	{attribute 'TcIecLibraryType'}
	{attribute 'external_name' := 'F_VN_StartAbsWatchdog_GUID_CDB36576_3437_07D6_675F_669467F27649'}
	(* Starts a cooperative watchdog given an absolute stop time. *)
	FUNCTION F_VN_StartAbsWatchdog : HRESULT
	VAR_INPUT
		tStop	:	DINT;	(* Stop time in us *)
		hrPrev	:	HRESULT;	(* HRESULT indicating the result of previous operations (If SUCCEEDED(hrPrev) equals false, no operation is executed.) *)
	END_VAR

END_FUNCTION

// Functions/Control Functions/F_VN_StartAbsWatchdogExp

	{attribute 'TcIecLibraryType'}
	{attribute 'external_name' := 'F_VN_StartAbsWatchdogExp_GUID_5DF99523_737E_0B42_4AEA_F8C27544139F'}
	(* Start a cooperative watchdog given an absolute stop time. (expert function) *)
	FUNCTION F_VN_StartAbsWatchdogExp : HRESULT
	VAR_INPUT
		tStop	:	DINT;	(* Stop time in us *)
		eWatchdogAccType	:	ETcWatchdogAccumulationType;	(* Accumalation method used for combining the results of multiple functions enclosed by this watchdog *)
		hrPrev	:	HRESULT;	(* HRESULT indicating the result of previous operations (If SUCCEEDED(hrPrev) equals false, no operation is executed.) *)
	END_VAR

END_FUNCTION

// Functions/Control Functions/F_VN_StartRelWatchdog

	{attribute 'TcIecLibraryType'}
	{attribute 'external_name' := 'F_VN_StartRelWatchdog_GUID_36307EEF_0607_0986_40C6_26A6AD435D06'}
	(* Starts a cooperative watchdog given a stop time relative to the current time. *)
	FUNCTION F_VN_StartRelWatchdog : HRESULT
	VAR_INPUT
		tStop	:	DINT;	(* Stop time in us *)
		hrPrev	:	HRESULT;	(* HRESULT indicating the result of previous operations (If SUCCEEDED(hrPrev) equals false, no operation is executed.) *)
	END_VAR

END_FUNCTION

// Functions/Control Functions/F_VN_StartRelWatchdogExp

	{attribute 'TcIecLibraryType'}
	{attribute 'external_name' := 'F_VN_StartRelWatchdogExp_GUID_3570B399_84A1_03B6_6569_A22DA832851F'}
	(* Start a cooperative watchdog given a stop time relative to the current time. (expert function) *)
	FUNCTION F_VN_StartRelWatchdogExp : HRESULT
	VAR_INPUT
		tStop	:	DINT;	(* Stop time in us *)
		eWatchdogAccType	:	ETcWatchdogAccumulationType;	(* Accumalation method used for combining the results of multiple functions enclosed by this watchdog *)
		hrPrev	:	HRESULT;	(* HRESULT indicating the result of previous operations (If SUCCEEDED(hrPrev) equals false, no operation is executed.) *)
	END_VAR

END_FUNCTION

// Functions/Control Functions/F_VN_StopWatchdog

	{attribute 'TcIecLibraryType'}
	{attribute 'external_name' := 'F_VN_StopWatchdog_GUID_5FE8103F_689C_0837_5C85_B4C88911468C'}
	(* Stops a watchdog and provide runtime information. *)
	FUNCTION F_VN_StopWatchdog : HRESULT
	VAR_INPUT
		hrStartWatchdog	:	HRESULT;	(* HRESULT indicating the result of the function used to start the watchdog (If SUCCEEDED(hrStartWatchdog) equals false, no operation is executed.) *)
	END_VAR
	VAR_OUTPUT
		nFunctionsMonitored	:	ULINT;	(* Returns the number of functions monitored *)
		nFractionProcessed	:	UDINT;	(* Returns the fraction processed accumulated over the monitored functions in percent *)
		tRest	:	DINT;	(* Returns the remaining computation time in us (may be negative) *)
	END_VAR

END_FUNCTION

// Functions/Image Segmentation/F_VN_AdaptiveThreshold

	{attribute 'TcIecLibraryType'}
	{attribute 'external_name' := 'F_VN_AdaptiveThreshold_GUID_B1BC4894_E3E4_011A_5395_9D7E3F472C15'}
	(* Apply an adaptive threshold to a gray level image. *)
	FUNCTION F_VN_AdaptiveThreshold : HRESULT
	VAR_INPUT
		ipSrcImage	:	ITcVnImage;	(* Source image (1 channel, elements of type USINT) *)
		ipDestImage	:	REFERENCE TO ITcVnImage;	(* Destination image (An appropriate destination image will be created if required.) *)
		fMaxValue	:	LREAL;	(* Value assigned to pixels for which the threshold condition is true *)
		hrPrev	:	HRESULT;	(* HRESULT indicating the result of previous operations (If SUCCEEDED(hrPrev) equals false, no operation is executed.) *)
	END_VAR

END_FUNCTION

// Functions/Image Segmentation/F_VN_AdaptiveThresholdExp

	{attribute 'TcIecLibraryType'}
	{attribute 'external_name' := 'F_VN_AdaptiveThresholdExp_GUID_E41ECDB8_1C09_051C_54A7_3EA4088C1F31'}
	(* Apply an adaptive threshold to a gray level image. (expert function) *)
	FUNCTION F_VN_AdaptiveThresholdExp : HRESULT
	VAR_INPUT
		ipSrcImage	:	ITcVnImage;	(* Source image (1 channel, elements of type USINT) *)
		ipDestImage	:	REFERENCE TO ITcVnImage;	(* Destination image (An appropriate destination image will be created if required.) *)
		fMaxValue	:	LREAL;	(* Value assigned to pixels for which the threshold condition is true *)
		eAdaptiveMethod	:	ETcVnAdaptiveThresholdMethod;	(* Adaptive threshold method to be applied (MEAN: threshold value will be calculated as a mean of the nBlockSize x nBlockSize neighborhood of (x,y) minus fConstant. GAUSSIAN: threshold value is a weighted sum (cross-correlation with a Gaussian window) of the nBlockSize x nBlockSize neighborhood of (x,y) minus fConstant. *)
		eThresholdType	:	ETcVnThresholdType;	(* Threshold type to be applied (only BINARY and BINARY_INV are supported) *)
		nBlockSize	:	UDINT;	(* Size of the pixel neighborhood to calculate the local threshold (3, 5, 7, ...) *)
		fConstant	:	LREAL;	(* Constant that is subtracted from the weighted mean of the pixel neighborhood, which leads to the local threshold *)
		hrPrev	:	HRESULT;	(* HRESULT indicating the result of previous operations (If SUCCEEDED(hrPrev) equals false, no operation is executed.) *)
	END_VAR

END_FUNCTION

// Functions/Image Segmentation/F_VN_CheckColorRange

	{attribute 'TcIecLibraryType'}
	{attribute 'external_name' := 'F_VN_CheckColorRange_GUID_5F05A5F1_5853_0BB7_40B0_9B84FD8E7D5D'}
	(* Check if the pixel values of an image lie in a given range. The destination image has the same size as the source image but only one channel with
          a pixel element size of 8 bit. Its elements are set to 255 if the corresponding pixels of the source image are in the checked range and set to 0 otherwise. *)
	FUNCTION F_VN_CheckColorRange : HRESULT
	VAR_INPUT
		ipSrcImage	:	ITcVnImage;	(* Source image *)
		ipDestImage	:	REFERENCE TO ITcVnImage;	(* Destination image (An appropriate destination image will be created if required.) *)
		aLowerBounds	:	REFERENCE TO TcVnVector4_LREAL;	(* Channel-wise lower bounds (Unused channels are ignored.) *)
		aUpperBounds	:	REFERENCE TO TcVnVector4_LREAL;	(* Channel-wise upper bounds (Unused channels are ignored.) *)
		hrPrev	:	HRESULT;	(* HRESULT indicating the result of previous operations (If SUCCEEDED(hrPrev) equals false, no operation is executed.) *)
	END_VAR

END_FUNCTION

// Functions/Image Segmentation/F_VN_Threshold

	{attribute 'TcIecLibraryType'}
	{attribute 'external_name' := 'F_VN_Threshold_GUID_F4BFB9FB_0241_0ABA_6497_302E4CB6A3F0'}
	(* Apply a fixed threshold or a dynamic threshold according to Otsu. *)
	FUNCTION F_VN_Threshold : HRESULT
	VAR_INPUT
		ipSrcImage	:	ITcVnImage;	(* Source image (For Otsu and Triangle threshold types, only 1 channel of TCVN_ET_USINT is supported) *)
		ipDestImage	:	REFERENCE TO ITcVnImage;	(* Destination image (An appropriate destination image will be created if required.) *)
		fThreshold	:	LREAL;	(* Fixed threshold (unused if dynamic thresholding is selected) *)
		fMaxValue	:	LREAL;	(* Maximum pixel value *)
		eThresholdType	:	ETcVnThresholdType;	(* Threshold type to be applied *)
		hrPrev	:	HRESULT;	(* HRESULT indicating the result of previous operations (If SUCCEEDED(hrPrev) equals false, no operation is executed.) *)
	END_VAR

END_FUNCTION

// Functions/Image Segmentation/F_VN_WatershedSegmentationExp

	{attribute 'TcIecLibraryType'}
	{attribute 'external_name' := 'F_VN_WatershedSegmentationExp_GUID_05447CF8_8CF8_0191_6A21_DD063D69ABC3'}
	(* Apply a marker-based watershed segmentation. (expert function) *)
	FUNCTION F_VN_WatershedSegmentationExp : HRESULT
	VAR_INPUT
		ipSrcImage	:	ITcVnImage;	(* Source image (USINT, 3 channels) *)
		ipDestImage	:	REFERENCE TO ITcVnImage;	(* Destination image (DINT, 1 channel. An appropriate image will be created if required.) *)
		ipMarkers	:	ITcVnImage;	(* Marker image (DINT, 1 channel) *)
		hrPrev	:	HRESULT;	(* HRESULT indicating the result of previous operations (If SUCCEEDED(hrPrev) equals false, no operation is executed.) *)
	END_VAR

END_FUNCTION

// Functions/Algebraic Container Operations/F_VN_AddContainers

	{attribute 'TcIecLibraryType'}
	{attribute 'external_name' := 'F_VN_AddContainers_GUID_34C85C3E_C161_0A16_51C0_0BD519308179'}
	(* Element-wise addition of two containers (same length and type). *)
	FUNCTION F_VN_AddContainers : HRESULT
	VAR_INPUT
		ipSrcContainer1	:	ITcVnContainer;	(* Source container 1 *)
		ipSrcContainer2	:	ITcVnContainer;	(* Source container 2 *)
		ipDestContainer	:	REFERENCE TO ITcVnContainer;	(* Returns the resulting container *)
		hrPrev	:	HRESULT;	(* HRESULT indicating the result of previous operations (If SUCCEEDED(hrPrev) equals false, no operation is executed.) *)
	END_VAR

END_FUNCTION

// Functions/Algebraic Container Operations/F_VN_BitwiseAndContainers

	{attribute 'TcIecLibraryType'}
	{attribute 'external_name' := 'F_VN_BitwiseAndContainers_GUID_EB7545F4_E7C1_0AC8_4065_DD74452EA045'}
	(* Element-wise application of a bit-wise AND operator to two containers (same length and type, integer only). *)
	FUNCTION F_VN_BitwiseAndContainers : HRESULT
	VAR_INPUT
		ipSrcContainer1	:	ITcVnContainer;	(* Source container 1 *)
		ipSrcContainer2	:	ITcVnContainer;	(* Source container 2 *)
		ipDestContainer	:	REFERENCE TO ITcVnContainer;	(* Returns the resulting container *)
		hrPrev	:	HRESULT;	(* HRESULT indicating the result of previous operations (If SUCCEEDED(hrPrev) equals false, no operation is executed.) *)
	END_VAR

END_FUNCTION

// Functions/Algebraic Container Operations/F_VN_BitwiseNotContainer

	{attribute 'TcIecLibraryType'}
	{attribute 'external_name' := 'F_VN_BitwiseNotContainer_GUID_F7145E10_2EC4_02FB_47B2_0962C0E72D64'}
	(* Element-wise application of a bit-wise NOT operator to a container (integer only). *)
	FUNCTION F_VN_BitwiseNotContainer : HRESULT
	VAR_INPUT
		ipSrcContainer	:	ITcVnContainer;	(* Source container *)
		ipDestContainer	:	REFERENCE TO ITcVnContainer;	(* Returns the resulting container *)
		hrPrev	:	HRESULT;	(* HRESULT indicating the result of previous operations (If SUCCEEDED(hrPrev) equals false, no operation is executed.) *)
	END_VAR

END_FUNCTION

// Functions/Algebraic Container Operations/F_VN_BitwiseOrContainers

	{attribute 'TcIecLibraryType'}
	{attribute 'external_name' := 'F_VN_BitwiseOrContainers_GUID_F073C4C8_8568_027C_57D8_3DAA401B2897'}
	(* Element-wise application of a bit-wise OR operator to two containers (same length and type, integer only). *)
	FUNCTION F_VN_BitwiseOrContainers : HRESULT
	VAR_INPUT
		ipSrcContainer1	:	ITcVnContainer;	(* Source container 1 *)
		ipSrcContainer2	:	ITcVnContainer;	(* Source container 2 *)
		ipDestContainer	:	REFERENCE TO ITcVnContainer;	(* Returns the resulting container *)
		hrPrev	:	HRESULT;	(* HRESULT indicating the result of previous operations (If SUCCEEDED(hrPrev) equals false, no operation is executed.) *)
	END_VAR

END_FUNCTION

// Functions/Algebraic Container Operations/F_VN_BitwiseXorContainers

	{attribute 'TcIecLibraryType'}
	{attribute 'external_name' := 'F_VN_BitwiseXorContainers_GUID_B00A3AA9_EBBD_07B2_4D65_1CE7DD68EA4F'}
	(* Element-wise application of a bit-wise XOR operator to two containers (same length and type, integer only). *)
	FUNCTION F_VN_BitwiseXorContainers : HRESULT
	VAR_INPUT
		ipSrcContainer1	:	ITcVnContainer;	(* Source container 1 *)
		ipSrcContainer2	:	ITcVnContainer;	(* Source container 2 *)
		ipDestContainer	:	REFERENCE TO ITcVnContainer;	(* Returns the resulting container *)
		hrPrev	:	HRESULT;	(* HRESULT indicating the result of previous operations (If SUCCEEDED(hrPrev) equals false, no operation is executed.) *)
	END_VAR

END_FUNCTION

// Functions/Algebraic Container Operations/F_VN_DivideContainers

	{attribute 'TcIecLibraryType'}
	{attribute 'external_name' := 'F_VN_DivideContainers_GUID_4F7AC07C_47AD_08DA_5AD8_2625E1B3B314'}
	(* Element-wise division of two containers (same length and type). In case of integer division by zero, the resulting element is set to 0 and S_DIVISION_BY_ZERO is returned instead of S_OK (value can be changed in F_VN_DivideContainersExp). *)
	FUNCTION F_VN_DivideContainers : HRESULT
	VAR_INPUT
		ipSrcContainer1	:	ITcVnContainer;	(* Source container 1 *)
		ipSrcContainer2	:	ITcVnContainer;	(* Source container 2 *)
		ipDestContainer	:	REFERENCE TO ITcVnContainer;	(* Returns the resulting container *)
		hrPrev	:	HRESULT;	(* HRESULT indicating the result of previous operations (If SUCCEEDED(hrPrev) equals false, no operation is executed.) *)
	END_VAR

END_FUNCTION

// Functions/Algebraic Container Operations/F_VN_DivideContainersExp

	{attribute 'TcIecLibraryType'}
	{attribute 'external_name' := 'F_VN_DivideContainersExp_GUID_5767066E_850E_06F8_62BD_9A0AC67D0659'}
	(* Element-wise division of two containers (same length and type). In case of integer division by zero, the resulting element is set to nIntDivideByZeroResult and S_DIVISION_BY_ZERO is returned instead of S_OK. (expert function) *)
	FUNCTION F_VN_DivideContainersExp : HRESULT
	VAR_INPUT
		ipSrcContainer1	:	ITcVnContainer;	(* Source container 1 *)
		ipSrcContainer2	:	ITcVnContainer;	(* Source container 2 *)
		ipDestContainer	:	REFERENCE TO ITcVnContainer;	(* Returns the resulting container *)
		nIntDivideByZeroResult	:	LINT;	(* Value set as result in case of integer division by zero *)
		hrPrev	:	HRESULT;	(* HRESULT indicating the result of previous operations (If SUCCEEDED(hrPrev) equals false, no operation is executed.) *)
	END_VAR

END_FUNCTION

// Functions/Algebraic Container Operations/F_VN_MaxContainer

	{attribute 'TcIecLibraryType'}
	{attribute 'external_name' := 'F_VN_MaxContainer_GUID_87E7AEC3_5BFE_0491_5BC1_F09A57C7AABE'}
	(* Element-wise maximum of two containers (same length and type). *)
	FUNCTION F_VN_MaxContainer : HRESULT
	VAR_INPUT
		ipSrcContainer1	:	ITcVnContainer;	(* Source container 1 *)
		ipSrcContainer2	:	ITcVnContainer;	(* Source container 2 *)
		ipDestContainer	:	REFERENCE TO ITcVnContainer;	(* Returns the resulting container *)
		hrPrev	:	HRESULT;	(* HRESULT indicating the result of previous operations (If SUCCEEDED(hrPrev) equals false, no operation is executed.) *)
	END_VAR

END_FUNCTION

// Functions/Algebraic Container Operations/F_VN_MinContainer

	{attribute 'TcIecLibraryType'}
	{attribute 'external_name' := 'F_VN_MinContainer_GUID_0D863741_BE56_02F1_6003_DB8B8D53248A'}
	(* Element-wise minimum of two containers (same length and type). *)
	FUNCTION F_VN_MinContainer : HRESULT
	VAR_INPUT
		ipSrcContainer1	:	ITcVnContainer;	(* Source container 1 *)
		ipSrcContainer2	:	ITcVnContainer;	(* Source container 2 *)
		ipDestContainer	:	REFERENCE TO ITcVnContainer;	(* Returns the resulting container *)
		hrPrev	:	HRESULT;	(* HRESULT indicating the result of previous operations (If SUCCEEDED(hrPrev) equals false, no operation is executed.) *)
	END_VAR

END_FUNCTION

// Functions/Algebraic Container Operations/F_VN_MultiplyContainers

	{attribute 'TcIecLibraryType'}
	{attribute 'external_name' := 'F_VN_MultiplyContainers_GUID_153C28CA_3B73_0635_5A9B_D25E4649912F'}
	(* Element-wise multiplication of two containers (same length and type). *)
	FUNCTION F_VN_MultiplyContainers : HRESULT
	VAR_INPUT
		ipSrcContainer1	:	ITcVnContainer;	(* Source container 1 *)
		ipSrcContainer2	:	ITcVnContainer;	(* Source container 2 *)
		ipDestContainer	:	REFERENCE TO ITcVnContainer;	(* Returns the resulting container *)
		hrPrev	:	HRESULT;	(* HRESULT indicating the result of previous operations (If SUCCEEDED(hrPrev) equals false, no operation is executed.) *)
	END_VAR

END_FUNCTION

// Functions/Algebraic Container Operations/F_VN_MultiplyWithContainerElements1

	{attribute 'TcIecLibraryType'}
	{attribute 'external_name' := 'F_VN_MultiplyWithContainerElements1_GUID_3A4363C5_2F07_0665_4907_45FBEBB2E86A'}
	(* Multiply each container element with a value. *)
	FUNCTION F_VN_MultiplyWithContainerElements1 : HRESULT
	VAR_INPUT
		fValue	:	LREAL;	(* Value *)
		ipContainer	:	ITcVnContainer;	(* Container with 1-dimensional elements *)
		hrPrev	:	HRESULT;	(* HRESULT indicating the result of previous operations (If SUCCEEDED(hrPrev) equals false, no operation is executed.) *)
	END_VAR

END_FUNCTION

// Functions/Algebraic Container Operations/F_VN_MultiplyWithContainerElements2

	{attribute 'TcIecLibraryType'}
	{attribute 'external_name' := 'F_VN_MultiplyWithContainerElements2_GUID_B731BD42_B03A_09DD_69AE_DE1A542F5D97'}
	(* Multiply each container element with a value. *)
	FUNCTION F_VN_MultiplyWithContainerElements2 : HRESULT
	VAR_INPUT
		aValue	:	REFERENCE TO TcVnVector2_LREAL;	(* Value *)
		ipContainer	:	ITcVnContainer;	(* Container with 2-dimensional elements *)
		hrPrev	:	HRESULT;	(* HRESULT indicating the result of previous operations (If SUCCEEDED(hrPrev) equals false, no operation is executed.) *)
	END_VAR

END_FUNCTION

// Functions/Algebraic Container Operations/F_VN_MultiplyWithContainerElements3

	{attribute 'TcIecLibraryType'}
	{attribute 'external_name' := 'F_VN_MultiplyWithContainerElements3_GUID_1C560529_161A_01EE_65F6_90383341846A'}
	(* Multiply each container element with a value. *)
	FUNCTION F_VN_MultiplyWithContainerElements3 : HRESULT
	VAR_INPUT
		aValue	:	REFERENCE TO TcVnVector3_LREAL;	(* Value *)
		ipContainer	:	ITcVnContainer;	(* Container with 3-dimensional elements *)
		hrPrev	:	HRESULT;	(* HRESULT indicating the result of previous operations (If SUCCEEDED(hrPrev) equals false, no operation is executed.) *)
	END_VAR

END_FUNCTION

// Functions/Algebraic Container Operations/F_VN_MultiplyWithContainerElements4

	{attribute 'TcIecLibraryType'}
	{attribute 'external_name' := 'F_VN_MultiplyWithContainerElements4_GUID_DD853A1D_EFF3_096A_6227_1AB3F2B2F982'}
	(* Multiply each container element with a value. *)
	FUNCTION F_VN_MultiplyWithContainerElements4 : HRESULT
	VAR_INPUT
		aValue	:	REFERENCE TO TcVnVector4_LREAL;	(* Value *)
		ipContainer	:	ITcVnContainer;	(* Container with 4-dimensional elements *)
		hrPrev	:	HRESULT;	(* HRESULT indicating the result of previous operations (If SUCCEEDED(hrPrev) equals false, no operation is executed.) *)
	END_VAR

END_FUNCTION

// Functions/Algebraic Container Operations/F_VN_NegateContainer

	{attribute 'TcIecLibraryType'}
	{attribute 'external_name' := 'F_VN_NegateContainer_GUID_07E50309_52EF_0D4D_4B31_50D2DD9AE529'}
	(* Element-wise negation of a container (two's complement). *)
	FUNCTION F_VN_NegateContainer : HRESULT
	VAR_INPUT
		ipSrcContainer	:	ITcVnContainer;	(* Source container *)
		ipDestContainer	:	REFERENCE TO ITcVnContainer;	(* Returns the resulting container (same type as ipSrcContainer) *)
		hrPrev	:	HRESULT;	(* HRESULT indicating the result of previous operations (If SUCCEEDED(hrPrev) equals false, no operation is executed.) *)
	END_VAR

END_FUNCTION

// Functions/Algebraic Container Operations/F_VN_SubtractContainers

	{attribute 'TcIecLibraryType'}
	{attribute 'external_name' := 'F_VN_SubtractContainers_GUID_2DA9CA96_A5D9_0422_5654_1161CA9C4960'}
	(* Element-wise subtraction of two containers (same length and type). *)
	FUNCTION F_VN_SubtractContainers : HRESULT
	VAR_INPUT
		ipSrcContainer1	:	ITcVnContainer;	(* Source container 1 *)
		ipSrcContainer2	:	ITcVnContainer;	(* Source container 2 *)
		ipDestContainer	:	REFERENCE TO ITcVnContainer;	(* Returns the resulting container *)
		hrPrev	:	HRESULT;	(* HRESULT indicating the result of previous operations (If SUCCEEDED(hrPrev) equals false, no operation is executed.) *)
	END_VAR

END_FUNCTION

// Functions/Algebraic Image Operations/F_VN_AddImages

	{attribute 'TcIecLibraryType'}
	{attribute 'external_name' := 'F_VN_AddImages_GUID_64CAC5EF_5C6A_0749_7465_A53EE4D2D5CD'}
	(* Element-wise addition of two images using saturation arithmetics. *)
	FUNCTION F_VN_AddImages : HRESULT
	VAR_INPUT
		ipSrcImage1	:	ITcVnImage;	(* First source image *)
		ipSrcImage2	:	ITcVnImage;	(* Second source image *)
		ipDestImage	:	REFERENCE TO ITcVnImage;	(* Destination image (An appropriate destination image will be created if required.) *)
		hrPrev	:	HRESULT;	(* HRESULT indicating the result of previous operations (If SUCCEEDED(hrPrev) equals false, no operation is executed.) *)
	END_VAR

END_FUNCTION

// Functions/Algebraic Image Operations/F_VN_AddImagesWeighted

	{attribute 'TcIecLibraryType'}
	{attribute 'external_name' := 'F_VN_AddImagesWeighted_GUID_685A3D3F_E01F_0D5D_7DEF_CD19484D6D9D'}
	(* Weighted, element-wise addition of two images using saturation arithmetics. *)
	FUNCTION F_VN_AddImagesWeighted : HRESULT
	VAR_INPUT
		ipSrcImage1	:	ITcVnImage;	(* First source image *)
		ipSrcImage2	:	ITcVnImage;	(* Second source image *)
		ipDestImage	:	REFERENCE TO ITcVnImage;	(* Destination image (An appropriate destination image will be created if required.) *)
		fWeight1	:	LREAL;	(* Weight factor applied to ipSrcImage1 *)
		fWeight2	:	LREAL;	(* Weight factor applied to ipSrcImage2 *)
		fDelta	:	LREAL;	(* Value added to the weighted sum of both images *)
		hrPrev	:	HRESULT;	(* HRESULT indicating the result of previous operations (If SUCCEEDED(hrPrev) equals false, no operation is executed.) *)
	END_VAR

END_FUNCTION

// Functions/Algebraic Image Operations/F_VN_AddImagesWeightedExp

	{attribute 'TcIecLibraryType'}
	{attribute 'external_name' := 'F_VN_AddImagesWeightedExp_GUID_B49E7431_16CC_0E7E_4344_6F996D6A935E'}
	(* Weighted, element-wise addition of two images using saturation arithmetics. *)
	FUNCTION F_VN_AddImagesWeightedExp : HRESULT
	VAR_INPUT
		ipSrcImage1	:	ITcVnImage;	(* First source image *)
		ipSrcImage2	:	ITcVnImage;	(* Second source image *)
		ipDestImage	:	REFERENCE TO ITcVnImage;	(* Destination image (An appropriate destination image will be created if required.) *)
		fWeight1	:	LREAL;	(* Weight factor applied to ipSrcImage1 *)
		fWeight2	:	LREAL;	(* Weight factor applied to ipSrcImage2 *)
		fDelta	:	LREAL;	(* Value added to the weighted sum of both images *)
		eDestType	:	ETcVnElementType;	(* Destination image depth *)
		hrPrev	:	HRESULT;	(* HRESULT indicating the result of previous operations (If SUCCEEDED(hrPrev) equals false, no operation is executed.) *)
	END_VAR

END_FUNCTION

// Functions/Algebraic Image Operations/F_VN_AddScalarToImage

	{attribute 'TcIecLibraryType'}
	{attribute 'external_name' := 'F_VN_AddScalarToImage_GUID_480F1A9E_1698_078E_60D8_B2611EBD2CE1'}
	(* Add a scalar value to each image pixel using saturation arithmetics. *)
	FUNCTION F_VN_AddScalarToImage : HRESULT
	VAR_INPUT
		fScalar	:	LREAL;	(* Scalar value *)
		ipSrcImage	:	ITcVnImage;	(* Source image *)
		ipDestImage	:	REFERENCE TO ITcVnImage;	(* Destination image (An appropriate destination image will be created if required.) *)
		hrPrev	:	HRESULT;	(* HRESULT indicating the result of previous operations (If SUCCEEDED(hrPrev) equals false, no operation is executed.) *)
	END_VAR

END_FUNCTION

// Functions/Algebraic Image Operations/F_VN_AddVectorToImage

	{attribute 'TcIecLibraryType'}
	{attribute 'external_name' := 'F_VN_AddVectorToImage_GUID_DD78328A_DF91_024C_6319_4FCE0B618763'}
	(* Add a vector (1 element for each image channel) to each image pixel using saturation arithmetics. *)
	FUNCTION F_VN_AddVectorToImage : HRESULT
	VAR_INPUT
		aVector	:	REFERENCE TO TcVnVector4_LREAL;	(* 4-element vector (1 element for each image channel. If the image has less channels, the further vector elements are ignored.) *)
		ipSrcImage	:	ITcVnImage;	(* Source image *)
		ipDestImage	:	REFERENCE TO ITcVnImage;	(* Destination image (An appropriate destination image will be created if required.) *)
		hrPrev	:	HRESULT;	(* HRESULT indicating the result of previous operations (If SUCCEEDED(hrPrev) equals false, no operation is executed.) *)
	END_VAR

END_FUNCTION

// Functions/Algebraic Image Operations/F_VN_BitwiseAndImages

	{attribute 'TcIecLibraryType'}
	{attribute 'external_name' := 'F_VN_BitwiseAndImages_GUID_BED381D7_0A5E_0CFE_7FFF_EA8B04927C22'}
	(* Element-wise application of a bit-wise AND operator to two images. *)
	FUNCTION F_VN_BitwiseAndImages : HRESULT
	VAR_INPUT
		ipSrcImage1	:	ITcVnImage;	(* First source image *)
		ipSrcImage2	:	ITcVnImage;	(* Second source image *)
		ipDestImage	:	REFERENCE TO ITcVnImage;	(* Destination image (An appropriate destination image will be created if required.) *)
		hrPrev	:	HRESULT;	(* HRESULT indicating the result of previous operations (If SUCCEEDED(hrPrev) equals false, no operation is executed.) *)
	END_VAR

END_FUNCTION

// Functions/Algebraic Image Operations/F_VN_BitwiseAndImagesExp

	{attribute 'TcIecLibraryType'}
	{attribute 'external_name' := 'F_VN_BitwiseAndImagesExp_GUID_28293BE7_304A_0FF6_4A33_EF5E74228BC5'}
	(* Element-wise application of a bit-wise AND operator to two images. (expert function) *)
	FUNCTION F_VN_BitwiseAndImagesExp : HRESULT
	VAR_INPUT
		ipSrcImage1	:	ITcVnImage;	(* First source image *)
		ipSrcImage2	:	ITcVnImage;	(* Second source image *)
		ipDestImage	:	REFERENCE TO ITcVnImage;	(* Destination image (An appropriate destination image will be created if required.) *)
		ipMask	:	ITcVnImage;	(* Mask to limit the operation to specific pixel positions (mask value 0: skip pixel, mask value > 0: apply operation to pixel) *)
		hrPrev	:	HRESULT;	(* HRESULT indicating the result of previous operations (If SUCCEEDED(hrPrev) equals false, no operation is executed.) *)
	END_VAR

END_FUNCTION

// Functions/Algebraic Image Operations/F_VN_BitwiseAndScalarWithImage

	{attribute 'TcIecLibraryType'}
	{attribute 'external_name' := 'F_VN_BitwiseAndScalarWithImage_GUID_385F968B_2133_03B0_6C50_EF84972C458A'}
	(* Bitwise and a scalar value with each image pixel. *)
	FUNCTION F_VN_BitwiseAndScalarWithImage : HRESULT
	VAR_INPUT
		fScalar	:	LREAL;	(* Scalar value *)
		ipSrcImage	:	ITcVnImage;	(* Source image *)
		ipDestImage	:	REFERENCE TO ITcVnImage;	(* Destination image (An appropriate destination image will be created if required.) *)
		hrPrev	:	HRESULT;	(* HRESULT indicating the result of previous operations (If SUCCEEDED(hrPrev) equals false, no operation is executed.) *)
	END_VAR

END_FUNCTION

// Functions/Algebraic Image Operations/F_VN_BitwiseAndVectorWithImage

	{attribute 'TcIecLibraryType'}
	{attribute 'external_name' := 'F_VN_BitwiseAndVectorWithImage_GUID_3C93DDCE_9C09_0A9B_53B4_AD9D39786D73'}
	(* Bitwise and a vector (1 element for each image channel) with each image pixel. *)
	FUNCTION F_VN_BitwiseAndVectorWithImage : HRESULT
	VAR_INPUT
		aVector	:	REFERENCE TO TcVnVector4_LREAL;	(* 4-element vector (1 element for each image channel. If the image has less channels, the further vector elements are ignored.) *)
		ipSrcImage	:	ITcVnImage;	(* Source image *)
		ipDestImage	:	REFERENCE TO ITcVnImage;	(* Destination image (An appropriate destination image will be created if required.) *)
		hrPrev	:	HRESULT;	(* HRESULT indicating the result of previous operations (If SUCCEEDED(hrPrev) equals false, no operation is executed.) *)
	END_VAR

END_FUNCTION

// Functions/Algebraic Image Operations/F_VN_BitwiseNotImage

	{attribute 'TcIecLibraryType'}
	{attribute 'external_name' := 'F_VN_BitwiseNotImage_GUID_0465B740_A753_018E_7A7A_2B6240A49397'}
	(* Element-wise application of a bit-wise NOT operator to an image. *)
	FUNCTION F_VN_BitwiseNotImage : HRESULT
	VAR_INPUT
		ipSrcImage	:	ITcVnImage;	(* Source image *)
		ipDestImage	:	REFERENCE TO ITcVnImage;	(* Destination image (An appropriate destination image will be created if required.) *)
		hrPrev	:	HRESULT;	(* HRESULT indicating the result of previous operations (If SUCCEEDED(hrPrev) equals false, no operation is executed.) *)
	END_VAR

END_FUNCTION

// Functions/Algebraic Image Operations/F_VN_BitwiseNotImageExp

	{attribute 'TcIecLibraryType'}
	{attribute 'external_name' := 'F_VN_BitwiseNotImageExp_GUID_3A1A5C98_D96F_0E1C_4FF5_B0411F693A04'}
	(* Element-wise application of a bit-wise NOT operator to an image. (expert function) *)
	FUNCTION F_VN_BitwiseNotImageExp : HRESULT
	VAR_INPUT
		ipSrcImage	:	ITcVnImage;	(* Source image *)
		ipDestImage	:	REFERENCE TO ITcVnImage;	(* Destination image (An appropriate destination image will be created if required.) *)
		ipMask	:	ITcVnImage;	(* Mask to limit the operation to specific pixel positions (mask value 0: skip pixel, mask value > 0: apply operation to pixel) *)
		hrPrev	:	HRESULT;	(* HRESULT indicating the result of previous operations (If SUCCEEDED(hrPrev) equals false, no operation is executed.) *)
	END_VAR

END_FUNCTION

// Functions/Algebraic Image Operations/F_VN_BitwiseOrImages

	{attribute 'TcIecLibraryType'}
	{attribute 'external_name' := 'F_VN_BitwiseOrImages_GUID_C9C88EF3_4746_03EA_5EC1_558B93379F53'}
	(* Element-wise application of a bit-wise OR operator to two images. *)
	FUNCTION F_VN_BitwiseOrImages : HRESULT
	VAR_INPUT
		ipSrcImage1	:	ITcVnImage;	(* First source image *)
		ipSrcImage2	:	ITcVnImage;	(* Second source image *)
		ipDestImage	:	REFERENCE TO ITcVnImage;	(* Destination image (An appropriate destination image will be created if required.) *)
		hrPrev	:	HRESULT;	(* HRESULT indicating the result of previous operations (If SUCCEEDED(hrPrev) equals false, no operation is executed.) *)
	END_VAR

END_FUNCTION

// Functions/Algebraic Image Operations/F_VN_BitwiseOrImagesExp

	{attribute 'TcIecLibraryType'}
	{attribute 'external_name' := 'F_VN_BitwiseOrImagesExp_GUID_6586601C_C1B5_0F53_55E7_A224AE8FCF5E'}
	(* Element-wise application of a bit-wise OR operator to two images. (expert function) *)
	FUNCTION F_VN_BitwiseOrImagesExp : HRESULT
	VAR_INPUT
		ipSrcImage1	:	ITcVnImage;	(* First source image *)
		ipSrcImage2	:	ITcVnImage;	(* Second source image *)
		ipDestImage	:	REFERENCE TO ITcVnImage;	(* Destination image (An appropriate destination image will be created if required.) *)
		ipMask	:	ITcVnImage;	(* Mask to limit the operation to specific pixel positions (mask value 0: skip pixel, mask value > 0: apply operation to pixel) *)
		hrPrev	:	HRESULT;	(* HRESULT indicating the result of previous operations (If SUCCEEDED(hrPrev) equals false, no operation is executed.) *)
	END_VAR

END_FUNCTION

// Functions/Algebraic Image Operations/F_VN_BitwiseOrScalarWithImage

	{attribute 'TcIecLibraryType'}
	{attribute 'external_name' := 'F_VN_BitwiseOrScalarWithImage_GUID_0F4D02C4_C8A2_00FD_49DB_E18AB49448D9'}
	(* Bitwise or a scalar value with each image pixel. *)
	FUNCTION F_VN_BitwiseOrScalarWithImage : HRESULT
	VAR_INPUT
		fScalar	:	LREAL;	(* Scalar value *)
		ipSrcImage	:	ITcVnImage;	(* Source image *)
		ipDestImage	:	REFERENCE TO ITcVnImage;	(* Destination image (An appropriate destination image will be created if required.) *)
		hrPrev	:	HRESULT;	(* HRESULT indicating the result of previous operations (If SUCCEEDED(hrPrev) equals false, no operation is executed.) *)
	END_VAR

END_FUNCTION

// Functions/Algebraic Image Operations/F_VN_BitwiseOrVectorWithImage

	{attribute 'TcIecLibraryType'}
	{attribute 'external_name' := 'F_VN_BitwiseOrVectorWithImage_GUID_489587CD_1238_0DA1_6B25_7D1344BACD7C'}
	(* Bitwise or a vector (1 element for each image channel) with each image pixel. *)
	FUNCTION F_VN_BitwiseOrVectorWithImage : HRESULT
	VAR_INPUT
		aVector	:	REFERENCE TO TcVnVector4_LREAL;	(* 4-element vector (1 element for each image channel. If the image has less channels, the further vector elements are ignored.) *)
		ipSrcImage	:	ITcVnImage;	(* Source image *)
		ipDestImage	:	REFERENCE TO ITcVnImage;	(* Destination image (An appropriate destination image will be created if required.) *)
		hrPrev	:	HRESULT;	(* HRESULT indicating the result of previous operations (If SUCCEEDED(hrPrev) equals false, no operation is executed.) *)
	END_VAR

END_FUNCTION

// Functions/Algebraic Image Operations/F_VN_BitwiseXorImages

	{attribute 'TcIecLibraryType'}
	{attribute 'external_name' := 'F_VN_BitwiseXorImages_GUID_087088B9_B544_039E_54C2_71F14D64B486'}
	(* Element-wise application of a bit-wise XOR operator to two images. *)
	FUNCTION F_VN_BitwiseXorImages : HRESULT
	VAR_INPUT
		ipSrcImage1	:	ITcVnImage;	(* First source image *)
		ipSrcImage2	:	ITcVnImage;	(* Second source image *)
		ipDestImage	:	REFERENCE TO ITcVnImage;	(* Destination image (An appropriate destination image will be created if required.) *)
		hrPrev	:	HRESULT;	(* HRESULT indicating the result of previous operations (If SUCCEEDED(hrPrev) equals false, no operation is executed.) *)
	END_VAR

END_FUNCTION

// Functions/Algebraic Image Operations/F_VN_BitwiseXorImagesExp

	{attribute 'TcIecLibraryType'}
	{attribute 'external_name' := 'F_VN_BitwiseXorImagesExp_GUID_5B312643_F44D_058A_6121_1BC423AE0A57'}
	(* Element-wise application of a bit-wise XOR operator to two images. (expert function) *)
	FUNCTION F_VN_BitwiseXorImagesExp : HRESULT
	VAR_INPUT
		ipSrcImage1	:	ITcVnImage;	(* First source image *)
		ipSrcImage2	:	ITcVnImage;	(* Second source image *)
		ipDestImage	:	REFERENCE TO ITcVnImage;	(* Destination image (An appropriate destination image will be created if required.) *)
		ipMask	:	ITcVnImage;	(* Mask to limit the operation to specific pixel positions (mask value 0: skip pixel, mask value > 0: apply operation to pixel) *)
		hrPrev	:	HRESULT;	(* HRESULT indicating the result of previous operations (If SUCCEEDED(hrPrev) equals false, no operation is executed.) *)
	END_VAR

END_FUNCTION

// Functions/Algebraic Image Operations/F_VN_BitwiseXorScalarWithImage

	{attribute 'TcIecLibraryType'}
	{attribute 'external_name' := 'F_VN_BitwiseXorScalarWithImage_GUID_31B4CF2D_2ED0_04ED_732B_D0B662A35C38'}
	(* Bitwise xor a scalar value with each image pixel. *)
	FUNCTION F_VN_BitwiseXorScalarWithImage : HRESULT
	VAR_INPUT
		fScalar	:	LREAL;	(* Scalar value *)
		ipSrcImage	:	ITcVnImage;	(* Source image *)
		ipDestImage	:	REFERENCE TO ITcVnImage;	(* Destination image (An appropriate destination image will be created if required.) *)
		hrPrev	:	HRESULT;	(* HRESULT indicating the result of previous operations (If SUCCEEDED(hrPrev) equals false, no operation is executed.) *)
	END_VAR

END_FUNCTION

// Functions/Algebraic Image Operations/F_VN_BitwiseXorVectorWithImage

	{attribute 'TcIecLibraryType'}
	{attribute 'external_name' := 'F_VN_BitwiseXorVectorWithImage_GUID_B7C272C7_A3D7_0471_7761_D679D6A1E01F'}
	(* Bitwise xor a vector (1 element for each image channel) with each image pixel. *)
	FUNCTION F_VN_BitwiseXorVectorWithImage : HRESULT
	VAR_INPUT
		aVector	:	REFERENCE TO TcVnVector4_LREAL;	(* 4-element vector (1 element for each image channel. If the image has less channels, the further vector elements are ignored.) *)
		ipSrcImage	:	ITcVnImage;	(* Source image *)
		ipDestImage	:	REFERENCE TO ITcVnImage;	(* Destination image (An appropriate destination image will be created if required.) *)
		hrPrev	:	HRESULT;	(* HRESULT indicating the result of previous operations (If SUCCEEDED(hrPrev) equals false, no operation is executed.) *)
	END_VAR

END_FUNCTION

// Functions/Algebraic Image Operations/F_VN_BlendImages

	{attribute 'TcIecLibraryType'}
	{attribute 'external_name' := 'F_VN_BlendImages_GUID_D93A64D1_22E7_04E5_4A4E_52FD2ABCC00F'}
	(* Blends two images, i.e. dest = (src1 * weight1 + src2 * weight2) / (weight1 + weight2). *)
	FUNCTION F_VN_BlendImages : HRESULT
	VAR_INPUT
		ipSrcImage1	:	ITcVnImage;	(* First source image (ET_USINT or ET_REAL) *)
		ipSrcImage2	:	ITcVnImage;	(* Second source image (same type and size as ipSrcImage1) *)
		ipWeights1	:	ITcVnImage;	(* Weights for ipSrcImage1 (1 channel, ET_REAL) *)
		ipWeights2	:	ITcVnImage;	(* Weights for ipSrcImage2 (1 channel, ET_REAL) *)
		ipDestImage	:	REFERENCE TO ITcVnImage;	(* Destination image (An appropriate destination image will be created if required.) *)
		hrPrev	:	HRESULT;	(* HRESULT indicating the result of previous operations (If SUCCEEDED(hrPrev) equals false, no operation is executed.) *)
	END_VAR

END_FUNCTION

// Functions/Algebraic Image Operations/F_VN_DivideImageByScalar

	{attribute 'TcIecLibraryType'}
	{attribute 'external_name' := 'F_VN_DivideImageByScalar_GUID_187859C9_D1A2_0B0B_4022_EFD4E62E74D1'}
	(* Divide each image pixel by a scalar value using saturation arithmetics. *)
	FUNCTION F_VN_DivideImageByScalar : HRESULT
	VAR_INPUT
		ipSrcImage	:	ITcVnImage;	(* Source image *)
		fScalar	:	LREAL;	(* Scalar value *)
		ipDestImage	:	REFERENCE TO ITcVnImage;	(* Destination image (An appropriate destination image will be created if required.) *)
		hrPrev	:	HRESULT;	(* HRESULT indicating the result of previous operations (If SUCCEEDED(hrPrev) equals false, no operation is executed.) *)
	END_VAR

END_FUNCTION

// Functions/Algebraic Image Operations/F_VN_DivideImageByVector

	{attribute 'TcIecLibraryType'}
	{attribute 'external_name' := 'F_VN_DivideImageByVector_GUID_E887A75A_A124_06BD_42FF_2C1F0BCD4B99'}
	(* Divides each image pixel by a vector (1 element for each image channel) using saturation arithmetics. *)
	FUNCTION F_VN_DivideImageByVector : HRESULT
	VAR_INPUT
		ipSrcImage	:	ITcVnImage;	(* Source image *)
		aVector	:	REFERENCE TO TcVnVector4_LREAL;	(* 4-element vector (1 element for each image channel. If the image has less channels, the further vector elements are ignored.) *)
		ipDestImage	:	REFERENCE TO ITcVnImage;	(* Destination image (An appropriate destination image will be created if required.) *)
		hrPrev	:	HRESULT;	(* HRESULT indicating the result of previous operations (If SUCCEEDED(hrPrev) equals false, no operation is executed.) *)
	END_VAR

END_FUNCTION

// Functions/Algebraic Image Operations/F_VN_DivideImages

	{attribute 'TcIecLibraryType'}
	{attribute 'external_name' := 'F_VN_DivideImages_GUID_087305F1_2B67_023E_4F20_56B7D9BE8EA7'}
	(* Element-wise division of two images using saturation arithmetics. (A division by zero equals zero.) *)
	FUNCTION F_VN_DivideImages : HRESULT
	VAR_INPUT
		ipSrcImage1	:	ITcVnImage;	(* First source image (dividend) *)
		ipSrcImage2	:	ITcVnImage;	(* Second source image (divisor) *)
		ipDestImage	:	REFERENCE TO ITcVnImage;	(* Destination image (An appropriate destination image will be created if required.) *)
		hrPrev	:	HRESULT;	(* HRESULT indicating the result of previous operations (If SUCCEEDED(hrPrev) equals false, no operation is executed.) *)
	END_VAR

END_FUNCTION

// Functions/Algebraic Image Operations/F_VN_DivideScalarByImage

	{attribute 'TcIecLibraryType'}
	{attribute 'external_name' := 'F_VN_DivideScalarByImage_GUID_5B0639CC_E574_0EEE_7288_2590ED6C94F0'}
	(* Divides a scalar value by each image pixel using saturation arithmetics. *)
	FUNCTION F_VN_DivideScalarByImage : HRESULT
	VAR_INPUT
		fScalar	:	LREAL;	(* Scalar value *)
		ipSrcImage	:	ITcVnImage;	(* Source image *)
		ipDestImage	:	REFERENCE TO ITcVnImage;	(* Destination image (An appropriate destination image will be created if required.) *)
		hrPrev	:	HRESULT;	(* HRESULT indicating the result of previous operations (If SUCCEEDED(hrPrev) equals false, no operation is executed.) *)
	END_VAR

END_FUNCTION

// Functions/Algebraic Image Operations/F_VN_DivideVectorByImage

	{attribute 'TcIecLibraryType'}
	{attribute 'external_name' := 'F_VN_DivideVectorByImage_GUID_50235AA1_D3BA_0AE8_42C5_6381525C4968'}
	(* Divides a vector (1 element for each image channel) by each image pixel using saturation arithmetics. *)
	FUNCTION F_VN_DivideVectorByImage : HRESULT
	VAR_INPUT
		aVector	:	REFERENCE TO TcVnVector4_LREAL;	(* 4-element vector (1 element for each image channel. If the image has less channels, the further vector elements are ignored.) *)
		ipSrcImage	:	ITcVnImage;	(* Source image *)
		ipDestImage	:	REFERENCE TO ITcVnImage;	(* Destination image (An appropriate destination image will be created if required.) *)
		hrPrev	:	HRESULT;	(* HRESULT indicating the result of previous operations (If SUCCEEDED(hrPrev) equals false, no operation is executed.) *)
	END_VAR

END_FUNCTION

// Functions/Algebraic Image Operations/F_VN_ElementwiseExp

	{attribute 'TcIecLibraryType'}
	{attribute 'external_name' := 'F_VN_ElementwiseExp_GUID_72C880BB_CD15_0A3B_4404_8857E9393471'}
	(* Computes the natural exponent of each pixel value. *)
	FUNCTION F_VN_ElementwiseExp : HRESULT
	VAR_INPUT
		ipSrcImage	:	ITcVnImage;	(* Source image (REAL or LREAL) *)
		ipDestImage	:	REFERENCE TO ITcVnImage;	(* Destination image (Same type and size as ipSrcImage, an appropriate image will be created if required.) *)
		hrPrev	:	HRESULT;	(* HRESULT indicating the result of previous operations (If SUCCEEDED(hrPrev) equals false, no operation is executed.) *)
	END_VAR

END_FUNCTION

// Functions/Algebraic Image Operations/F_VN_ElementwiseLog

	{attribute 'TcIecLibraryType'}
	{attribute 'external_name' := 'F_VN_ElementwiseLog_GUID_6A1F9A82_6FBA_0C25_7DB0_453D95D27638'}
	(* Computes the natural logarithm of each pixel value. *)
	FUNCTION F_VN_ElementwiseLog : HRESULT
	VAR_INPUT
		ipSrcImage	:	ITcVnImage;	(* Source image (REAL or LREAL) *)
		ipDestImage	:	REFERENCE TO ITcVnImage;	(* Destination image (Same type and size as ipSrcImage, an appropriate image will be created if required.) *)
		hrPrev	:	HRESULT;	(* HRESULT indicating the result of previous operations (If SUCCEEDED(hrPrev) equals false, no operation is executed.) *)
	END_VAR

END_FUNCTION

// Functions/Algebraic Image Operations/F_VN_MaxImage

	{attribute 'TcIecLibraryType'}
	{attribute 'external_name' := 'F_VN_MaxImage_GUID_0A561FE2_31A1_08D1_7E19_47146405185D'}
	(* Element-wise maximum of two images. *)
	FUNCTION F_VN_MaxImage : HRESULT
	VAR_INPUT
		ipSrcImage1	:	ITcVnImage;	(* First source image *)
		ipSrcImage2	:	ITcVnImage;	(* Second source image *)
		ipDestImage	:	REFERENCE TO ITcVnImage;	(* Destination image (An appropriate destination image will be created if required.) *)
		hrPrev	:	HRESULT;	(* HRESULT indicating the result of previous operations (If SUCCEEDED(hrPrev) equals false, no operation is executed.) *)
	END_VAR

END_FUNCTION

// Functions/Algebraic Image Operations/F_VN_MaxImageExp

	{attribute 'TcIecLibraryType'}
	{attribute 'external_name' := 'F_VN_MaxImageExp_GUID_041B8AFF_FB90_0313_59DC_E9458C512885'}
	(* Element-wise maximum of two images. (expert function) *)
	FUNCTION F_VN_MaxImageExp : HRESULT
	VAR_INPUT
		ipSrcImage1	:	ITcVnImage;	(* First source image *)
		ipSrcImage2	:	ITcVnImage;	(* Second source image *)
		ipDestImage	:	REFERENCE TO ITcVnImage;	(* Destination image (An appropriate destination image will be created if required.) *)
		ipMask	:	ITcVnImage;	(* Mask of type USINT *)
		hrPrev	:	HRESULT;	(* HRESULT indicating the result of previous operations (If SUCCEEDED(hrPrev) equals false, no operation is executed.) *)
	END_VAR

END_FUNCTION

// Functions/Algebraic Image Operations/F_VN_MaxImageWithScalar

	{attribute 'TcIecLibraryType'}
	{attribute 'external_name' := 'F_VN_MaxImageWithScalar_GUID_5F966B15_938B_04A4_489E_3DBA85718489'}
	(* Element-wise maximum of image and scalar value. *)
	FUNCTION F_VN_MaxImageWithScalar : HRESULT
	VAR_INPUT
		fScalar	:	LREAL;	(* Scalar value *)
		ipSrcImage	:	ITcVnImage;	(* Source image *)
		ipDestImage	:	REFERENCE TO ITcVnImage;	(* Destination image (An appropriate destination image will be created if required.) *)
		hrPrev	:	HRESULT;	(* HRESULT indicating the result of previous operations (If SUCCEEDED(hrPrev) equals false, no operation is executed.) *)
	END_VAR

END_FUNCTION

// Functions/Algebraic Image Operations/F_VN_MaxImageWithScalarExp

	{attribute 'TcIecLibraryType'}
	{attribute 'external_name' := 'F_VN_MaxImageWithScalarExp_GUID_2FA5C0D8_7C09_0A64_4EF6_B4AF38F66D1B'}
	(* Element-wise maximum of image and scalar value. (expert function) *)
	FUNCTION F_VN_MaxImageWithScalarExp : HRESULT
	VAR_INPUT
		fScalar	:	LREAL;	(* Scalar value *)
		ipSrcImage	:	ITcVnImage;	(* Source image *)
		ipDestImage	:	REFERENCE TO ITcVnImage;	(* Destination image (An appropriate destination image will be created if required.) *)
		ipMask	:	ITcVnImage;	(* Mask of type USINT *)
		hrPrev	:	HRESULT;	(* HRESULT indicating the result of previous operations (If SUCCEEDED(hrPrev) equals false, no operation is executed.) *)
	END_VAR

END_FUNCTION

// Functions/Algebraic Image Operations/F_VN_MaxImageWithVector

	{attribute 'TcIecLibraryType'}
	{attribute 'external_name' := 'F_VN_MaxImageWithVector_GUID_BDE7E41A_4057_03E6_503C_8A6A3EBECEEA'}
	(* Element-wise maximum of image and vector (1 element for each image channel). *)
	FUNCTION F_VN_MaxImageWithVector : HRESULT
	VAR_INPUT
		aVector	:	REFERENCE TO TcVnVector4_LREAL;	(* 4-element vector (1 element for each image channel. If the image has less channels, the further vector elements are ignored.) *)
		ipSrcImage	:	ITcVnImage;	(* Source image *)
		ipDestImage	:	REFERENCE TO ITcVnImage;	(* Destination image (An appropriate destination image will be created if required.) *)
		hrPrev	:	HRESULT;	(* HRESULT indicating the result of previous operations (If SUCCEEDED(hrPrev) equals false, no operation is executed.) *)
	END_VAR

END_FUNCTION

// Functions/Algebraic Image Operations/F_VN_MaxImageWithVectorExp

	{attribute 'TcIecLibraryType'}
	{attribute 'external_name' := 'F_VN_MaxImageWithVectorExp_GUID_AD0A87D8_DF17_098C_5148_46940528F925'}
	(* Element-wise maximum of image and vector (1 element for each image channel). (expert function) *)
	FUNCTION F_VN_MaxImageWithVectorExp : HRESULT
	VAR_INPUT
		aVector	:	REFERENCE TO TcVnVector4_LREAL;	(* 4-element vector (1 element for each image channel. If the image has less channels, the further vector elements are ignored.) *)
		ipSrcImage	:	ITcVnImage;	(* Source image *)
		ipDestImage	:	REFERENCE TO ITcVnImage;	(* Destination image (An appropriate destination image will be created if required.) *)
		ipMask	:	ITcVnImage;	(* Mask of type USINT *)
		hrPrev	:	HRESULT;	(* HRESULT indicating the result of previous operations (If SUCCEEDED(hrPrev) equals false, no operation is executed.) *)
	END_VAR

END_FUNCTION

// Functions/Algebraic Image Operations/F_VN_MinImage

	{attribute 'TcIecLibraryType'}
	{attribute 'external_name' := 'F_VN_MinImage_GUID_6ACE3486_6C7A_0695_5558_66ACCAE437BA'}
	(* Element-wise minimum of two images. *)
	FUNCTION F_VN_MinImage : HRESULT
	VAR_INPUT
		ipSrcImage1	:	ITcVnImage;	(* First source image *)
		ipSrcImage2	:	ITcVnImage;	(* Second source image *)
		ipDestImage	:	REFERENCE TO ITcVnImage;	(* Destination image (An appropriate destination image will be created if required.) *)
		hrPrev	:	HRESULT;	(* HRESULT indicating the result of previous operations (If SUCCEEDED(hrPrev) equals false, no operation is executed.) *)
	END_VAR

END_FUNCTION

// Functions/Algebraic Image Operations/F_VN_MinImageExp

	{attribute 'TcIecLibraryType'}
	{attribute 'external_name' := 'F_VN_MinImageExp_GUID_8E0FEFA8_12AA_03C9_6011_18C80D5BE112'}
	(* Element-wise minimum of two images. (expert function) *)
	FUNCTION F_VN_MinImageExp : HRESULT
	VAR_INPUT
		ipSrcImage1	:	ITcVnImage;	(* First source image *)
		ipSrcImage2	:	ITcVnImage;	(* Second source image *)
		ipDestImage	:	REFERENCE TO ITcVnImage;	(* Destination image (An appropriate destination image will be created if required.) *)
		ipMask	:	ITcVnImage;	(* Mask of type USINT *)
		hrPrev	:	HRESULT;	(* HRESULT indicating the result of previous operations (If SUCCEEDED(hrPrev) equals false, no operation is executed.) *)
	END_VAR

END_FUNCTION

// Functions/Algebraic Image Operations/F_VN_MinImageWithScalar

	{attribute 'TcIecLibraryType'}
	{attribute 'external_name' := 'F_VN_MinImageWithScalar_GUID_871726C6_DE75_0088_7DB3_7D15AFBC38AF'}
	(* Element-wise minimum of image and scalar value. *)
	FUNCTION F_VN_MinImageWithScalar : HRESULT
	VAR_INPUT
		fScalar	:	LREAL;	(* Scalar value *)
		ipSrcImage	:	ITcVnImage;	(* Source image *)
		ipDestImage	:	REFERENCE TO ITcVnImage;	(* Destination image (An appropriate destination image will be created if required.) *)
		hrPrev	:	HRESULT;	(* HRESULT indicating the result of previous operations (If SUCCEEDED(hrPrev) equals false, no operation is executed.) *)
	END_VAR

END_FUNCTION

// Functions/Algebraic Image Operations/F_VN_MinImageWithScalarExp

	{attribute 'TcIecLibraryType'}
	{attribute 'external_name' := 'F_VN_MinImageWithScalarExp_GUID_42002185_56E8_0CA4_7C19_FA31CE9853EA'}
	(* Element-wise minimum of image and scalar value. (expert function) *)
	FUNCTION F_VN_MinImageWithScalarExp : HRESULT
	VAR_INPUT
		fScalar	:	LREAL;	(* Scalar value *)
		ipSrcImage	:	ITcVnImage;	(* Source image *)
		ipDestImage	:	REFERENCE TO ITcVnImage;	(* Destination image (An appropriate destination image will be created if required.) *)
		ipMask	:	ITcVnImage;	(* Mask of type USINT *)
		hrPrev	:	HRESULT;	(* HRESULT indicating the result of previous operations (If SUCCEEDED(hrPrev) equals false, no operation is executed.) *)
	END_VAR

END_FUNCTION

// Functions/Algebraic Image Operations/F_VN_MinImageWithVector

	{attribute 'TcIecLibraryType'}
	{attribute 'external_name' := 'F_VN_MinImageWithVector_GUID_A6DA65D7_CDD3_053D_6BEC_86E3208CE375'}
	(* Element-wise minimum of image and vector (1 element for each image channel). *)
	FUNCTION F_VN_MinImageWithVector : HRESULT
	VAR_INPUT
		aVector	:	REFERENCE TO TcVnVector4_LREAL;	(* 4-element vector (1 element for each image channel. If the image has less channels, the further vector elements are ignored.) *)
		ipSrcImage	:	ITcVnImage;	(* Source image *)
		ipDestImage	:	REFERENCE TO ITcVnImage;	(* Destination image (An appropriate destination image will be created if required.) *)
		hrPrev	:	HRESULT;	(* HRESULT indicating the result of previous operations (If SUCCEEDED(hrPrev) equals false, no operation is executed.) *)
	END_VAR

END_FUNCTION

// Functions/Algebraic Image Operations/F_VN_MinImageWithVectorExp

	{attribute 'TcIecLibraryType'}
	{attribute 'external_name' := 'F_VN_MinImageWithVectorExp_GUID_09B5E25E_4A03_0947_5FB7_01E46AB6EC60'}
	(* Element-wise minimum of image and vector (1 element for each image channel). (expert function) *)
	FUNCTION F_VN_MinImageWithVectorExp : HRESULT
	VAR_INPUT
		aVector	:	REFERENCE TO TcVnVector4_LREAL;	(* 4-element vector (1 element for each image channel. If the image has less channels, the further vector elements are ignored.) *)
		ipSrcImage	:	ITcVnImage;	(* Source image *)
		ipDestImage	:	REFERENCE TO ITcVnImage;	(* Destination image (An appropriate destination image will be created if required.) *)
		ipMask	:	ITcVnImage;	(* Mask of type USINT *)
		hrPrev	:	HRESULT;	(* HRESULT indicating the result of previous operations (If SUCCEEDED(hrPrev) equals false, no operation is executed.) *)
	END_VAR

END_FUNCTION

// Functions/Algebraic Image Operations/F_VN_MultiplyImages

	{attribute 'TcIecLibraryType'}
	{attribute 'external_name' := 'F_VN_MultiplyImages_GUID_F97D119F_8EA3_08EA_5265_7BF041F9E095'}
	(* Element-wise multiplication of two images using saturation arithmetics. *)
	FUNCTION F_VN_MultiplyImages : HRESULT
	VAR_INPUT
		ipSrcImage1	:	ITcVnImage;	(* First source image *)
		ipSrcImage2	:	ITcVnImage;	(* Second source image *)
		ipDestImage	:	REFERENCE TO ITcVnImage;	(* Destination image (An appropriate destination image will be created if required.) *)
		hrPrev	:	HRESULT;	(* HRESULT indicating the result of previous operations (If SUCCEEDED(hrPrev) equals false, no operation is executed.) *)
	END_VAR

END_FUNCTION

// Functions/Algebraic Image Operations/F_VN_MultiplyImageWithScalar

	{attribute 'TcIecLibraryType'}
	{attribute 'external_name' := 'F_VN_MultiplyImageWithScalar_GUID_CAFC6B2C_5602_048C_4EE3_5C2970962994'}
	(* Multiply each image pixel by a scalar value using saturation arithmetics. *)
	FUNCTION F_VN_MultiplyImageWithScalar : HRESULT
	VAR_INPUT
		fScalar	:	LREAL;	(* Scalar value *)
		ipSrcImage	:	ITcVnImage;	(* Source image *)
		ipDestImage	:	REFERENCE TO ITcVnImage;	(* Destination image (An appropriate destination image will be created if required.) *)
		hrPrev	:	HRESULT;	(* HRESULT indicating the result of previous operations (If SUCCEEDED(hrPrev) equals false, no operation is executed.) *)
	END_VAR

END_FUNCTION

// Functions/Algebraic Image Operations/F_VN_MultiplyImageWithVector

	{attribute 'TcIecLibraryType'}
	{attribute 'external_name' := 'F_VN_MultiplyImageWithVector_GUID_2181E52A_3854_03DE_7996_DDF7AFEEE3CC'}
	(* Multiply each image pixel by a vector (1 element for each image channel) using saturation arithmetics. *)
	FUNCTION F_VN_MultiplyImageWithVector : HRESULT
	VAR_INPUT
		aVector	:	REFERENCE TO TcVnVector4_LREAL;	(* 4-element vector (1 element for each image channel. If the image has less channels, the further vector elements are ignored.) *)
		ipSrcImage	:	ITcVnImage;	(* Source image *)
		ipDestImage	:	REFERENCE TO ITcVnImage;	(* Destination image (An appropriate destination image will be created if required.) *)
		hrPrev	:	HRESULT;	(* HRESULT indicating the result of previous operations (If SUCCEEDED(hrPrev) equals false, no operation is executed.) *)
	END_VAR

END_FUNCTION

// Functions/Algebraic Image Operations/F_VN_SubtractImageFromScalar

	{attribute 'TcIecLibraryType'}
	{attribute 'external_name' := 'F_VN_SubtractImageFromScalar_GUID_C37D6BD4_206D_0634_7DA5_7C245A64C5EF'}
	(* Subtract each image pixel from a scalar value using saturation arithmetics. *)
	FUNCTION F_VN_SubtractImageFromScalar : HRESULT
	VAR_INPUT
		fScalar	:	LREAL;	(* Scalar value *)
		ipSrcImage	:	ITcVnImage;	(* Source image *)
		ipDestImage	:	REFERENCE TO ITcVnImage;	(* Destination image (An appropriate destination image will be created if required.) *)
		hrPrev	:	HRESULT;	(* HRESULT indicating the result of previous operations (If SUCCEEDED(hrPrev) equals false, no operation is executed.) *)
	END_VAR

END_FUNCTION

// Functions/Algebraic Image Operations/F_VN_SubtractImageFromVector

	{attribute 'TcIecLibraryType'}
	{attribute 'external_name' := 'F_VN_SubtractImageFromVector_GUID_6C8636EB_C22B_0ACB_6CD1_AB08AB71902A'}
	(* Subtract each image pixel from a vector (1 element for each image channel) using saturation arithmetics. *)
	FUNCTION F_VN_SubtractImageFromVector : HRESULT
	VAR_INPUT
		aVector	:	REFERENCE TO TcVnVector4_LREAL;	(* 4-element vector (1 element for each image channel. If the image has less channels, the further vector elements are ignored.) *)
		ipSrcImage	:	ITcVnImage;	(* Source image *)
		ipDestImage	:	REFERENCE TO ITcVnImage;	(* Destination image (An appropriate destination image will be created if required.) *)
		hrPrev	:	HRESULT;	(* HRESULT indicating the result of previous operations (If SUCCEEDED(hrPrev) equals false, no operation is executed.) *)
	END_VAR

END_FUNCTION

// Functions/Algebraic Image Operations/F_VN_SubtractImages

	{attribute 'TcIecLibraryType'}
	{attribute 'external_name' := 'F_VN_SubtractImages_GUID_E87C6004_3B96_0E56_7E0B_3B3D0C2DD439'}
	(* Element-wise subtraction of two images using saturation arithmetics. *)
	FUNCTION F_VN_SubtractImages : HRESULT
	VAR_INPUT
		ipSrcImage1	:	ITcVnImage;	(* First source image (minuend) *)
		ipSrcImage2	:	ITcVnImage;	(* Second source image (subtrahend) *)
		ipDestImage	:	REFERENCE TO ITcVnImage;	(* Destination image (An appropriate destination image will be created if required.) *)
		hrPrev	:	HRESULT;	(* HRESULT indicating the result of previous operations (If SUCCEEDED(hrPrev) equals false, no operation is executed.) *)
	END_VAR

END_FUNCTION

// Functions/Algebraic Image Operations/F_VN_SubtractScalarFromImage

	{attribute 'TcIecLibraryType'}
	{attribute 'external_name' := 'F_VN_SubtractScalarFromImage_GUID_31A28C83_0D11_071A_614A_AF2228DB9ACD'}
	(* Subtract a scalar value from each image pixel using saturation arithmetics. *)
	FUNCTION F_VN_SubtractScalarFromImage : HRESULT
	VAR_INPUT
		ipSrcImage	:	ITcVnImage;	(* Source image *)
		fScalar	:	LREAL;	(* Scalar value *)
		ipDestImage	:	REFERENCE TO ITcVnImage;	(* Destination image (An appropriate destination image will be created if required.) *)
		hrPrev	:	HRESULT;	(* HRESULT indicating the result of previous operations (If SUCCEEDED(hrPrev) equals false, no operation is executed.) *)
	END_VAR

END_FUNCTION

// Functions/Algebraic Image Operations/F_VN_SubtractVectorFromImage

	{attribute 'TcIecLibraryType'}
	{attribute 'external_name' := 'F_VN_SubtractVectorFromImage_GUID_419244AF_B338_049D_6708_EC0EBE0CAEB6'}
	(* Subtract a vector (1 element for each image channel) from each image pixel using saturation arithmetics. *)
	FUNCTION F_VN_SubtractVectorFromImage : HRESULT
	VAR_INPUT
		ipSrcImage	:	ITcVnImage;	(* Source image *)
		aVector	:	REFERENCE TO TcVnVector4_LREAL;	(* 4-element vector (1 element for each image channel. If the image has less channels, the further vector elements are ignored.) *)
		ipDestImage	:	REFERENCE TO ITcVnImage;	(* Destination image (An appropriate destination image will be created if required.) *)
		hrPrev	:	HRESULT;	(* HRESULT indicating the result of previous operations (If SUCCEEDED(hrPrev) equals false, no operation is executed.) *)
	END_VAR

END_FUNCTION

// Functions/Image Analysis/F_VN_CannyEdgeDetection

	{attribute 'TcIecLibraryType'}
	{attribute 'external_name' := 'F_VN_CannyEdgeDetection_GUID_D6863D47_B135_01BE_6547_D47F8B6C73F8'}
	(* Find edges using the Canny edge detection algorithm. *)
	FUNCTION F_VN_CannyEdgeDetection : HRESULT
	VAR_INPUT
		ipSrcImage	:	ITcVnImage;	(* Source image (elements of type USINT) *)
		ipDestImage	:	REFERENCE TO ITcVnImage;	(* Destination image (elements of type USINT. An appropriate destination image will be created if required.) *)
		fThresholdLow	:	LREAL;	(* Low threshold *)
		fThresholdHigh	:	LREAL;	(* High threshold *)
		hrPrev	:	HRESULT;	(* HRESULT indicating the result of previous operations (If SUCCEEDED(hrPrev) equals false, no operation is executed.) *)
	END_VAR

END_FUNCTION

// Functions/Image Analysis/F_VN_CannyEdgeDetectionExp

	{attribute 'TcIecLibraryType'}
	{attribute 'external_name' := 'F_VN_CannyEdgeDetectionExp_GUID_16DFE865_409B_04D8_535E_0F9F3555FE96'}
	(* Find edges using the Canny edge detection algorithm. (expert function) *)
	FUNCTION F_VN_CannyEdgeDetectionExp : HRESULT
	VAR_INPUT
		ipSrcImage	:	ITcVnImage;	(* Source image (elements of type USINT) *)
		ipDestImage	:	REFERENCE TO ITcVnImage;	(* Destination image (elements of type USINT. An appropriate destination image will be created if required.) *)
		fThresholdLow	:	LREAL;	(* Low threshold *)
		fThresholdHigh	:	LREAL;	(* High threshold *)
		nApertureSize	:	UDINT;	(* Aperture size for the Sobel operator (3, 5, 7) *)
		bL2Gradient	:	BOOL;	(* If true, the more accurate (and slower) L2 norm is used instead of the L1 norm *)
		hrPrev	:	HRESULT;	(* HRESULT indicating the result of previous operations (If SUCCEEDED(hrPrev) equals false, no operation is executed.) *)
	END_VAR

END_FUNCTION

// Functions/Image Analysis/F_VN_ConnectedComponents

	{attribute 'TcIecLibraryType'}
	{attribute 'external_name' := 'F_VN_ConnectedComponents_GUID_184C9DF1_D88E_0FA8_78D5_15AC9D0988C9'}
	(* Computes the connected components of an image. *)
	FUNCTION F_VN_ConnectedComponents : HRESULT
	VAR_INPUT
		ipSrcImage	:	ITcVnImage;	(* Source image with threshold applied (1 channel, USINT) *)
		ipLabelImage	:	REFERENCE TO ITcVnImage;	(* Returns the labels for each source image pixel (1 channel, DINT. An appropriate destination image will be created if required.) *)
		nLabels	:	REFERENCE TO DINT;	(* Returns the number of labels *)
		hrPrev	:	HRESULT;	(* HRESULT indicating the result of previous operations (If SUCCEEDED(hrPrev) equals false, no operation is executed.) *)
	END_VAR

END_FUNCTION

// Functions/Image Analysis/F_VN_ConnectedComponentsExp

	{attribute 'TcIecLibraryType'}
	{attribute 'external_name' := 'F_VN_ConnectedComponentsExp_GUID_C0D13FA0_3691_0D18_7A93_42977985AEB5'}
	(* Computes the connected components of an image. (expert function) *)
	FUNCTION F_VN_ConnectedComponentsExp : HRESULT
	VAR_INPUT
		ipSrcImage	:	ITcVnImage;	(* Source image with threshold applied (1 channel, USINT) *)
		ipLabelImage	:	REFERENCE TO ITcVnImage;	(* Returns the labels for each source image pixel (1 channel, type depends on eLabelType. An appropriate destination image will be created if required.) *)
		nLabels	:	REFERENCE TO DINT;	(* Returns the number of labels *)
		eConnectivity	:	ETcVnPixelConnectivity;	(* Selects if 4- or 8-way pixel connectivity should be used *)
		eLabelType	:	ETcVnElementType;	(* Selects the type of ipLabelImage (only UINT or DINT supported) *)
		eAlgorithm	:	ETcVnConnectedComponentsAlgorithm;	(* Selects the applied algorithm *)
		hrPrev	:	HRESULT;	(* HRESULT indicating the result of previous operations (If SUCCEEDED(hrPrev) equals false, no operation is executed.) *)
	END_VAR

END_FUNCTION

// Functions/Image Analysis/F_VN_ConnectedComponentsWithStats

	{attribute 'TcIecLibraryType'}
	{attribute 'external_name' := 'F_VN_ConnectedComponentsWithStats_GUID_760805DD_7C9C_074B_7A25_2DBA54EA94C1'}
	(* Computes the connected components and corresponding statistics of an image. *)
	FUNCTION F_VN_ConnectedComponentsWithStats : HRESULT
	VAR_INPUT
		ipSrcImage	:	ITcVnImage;	(* Source image with threshold applied (1 channel, USINT) *)
		ipLabelImage	:	REFERENCE TO ITcVnImage;	(* Returns the labels for each source image pixel (1 channel, DINT. An appropriate destination image will be created if required.) *)
		ipBoundingBoxes	:	REFERENCE TO ITcVnContainer;	(* Returns the bounding boxes for each labeled region. (ContainerType_Vector_TcVnRectangle_DINT; Non-zero interface pointers are reused.) *)
		ipNumPixels	:	REFERENCE TO ITcVnContainer;	(* Returns the number of pixels for each labeled region. (ContainerType_Vector_DINT; Non-zero interface pointers are reused.) *)
		ipCentroids	:	REFERENCE TO ITcVnContainer;	(* Returns the centroids for each labeled region. (ContainerType_Vector_TcVnPoint2_LREAL; Non-zero interface pointers are reused.) *)
		nLabels	:	REFERENCE TO DINT;	(* Returns the number of labels *)
		hrPrev	:	HRESULT;	(* HRESULT indicating the result of previous operations (If SUCCEEDED(hrPrev) equals false, no operation is executed.) *)
	END_VAR

END_FUNCTION

// Functions/Image Analysis/F_VN_ConnectedComponentsWithStatsExp

	{attribute 'TcIecLibraryType'}
	{attribute 'external_name' := 'F_VN_ConnectedComponentsWithStatsExp_GUID_BE1EA54B_7DCB_09A5_59BB_23F867F837B9'}
	(* Computes the connected components and corresponding statistics of an image. (expert function) *)
	FUNCTION F_VN_ConnectedComponentsWithStatsExp : HRESULT
	VAR_INPUT
		ipSrcImage	:	ITcVnImage;	(* Source image with threshold applied (1 channel, USINT) *)
		ipLabelImage	:	REFERENCE TO ITcVnImage;	(* Returns the labels for each source image pixel (1 channel, DINT. An appropriate destination image will be created if required.) *)
		ipBoundingBoxes	:	REFERENCE TO ITcVnContainer;	(* Returns the bounding boxes for each labeled region. (ContainerType_Vector_TcVnRectangle_DINT; Non-zero interface pointers are reused.) *)
		ipNumPixels	:	REFERENCE TO ITcVnContainer;	(* Returns the number of pixels for each labeled region. (ContainerType_Vector_DINT; Non-zero interface pointers are reused.) *)
		ipCentroids	:	REFERENCE TO ITcVnContainer;	(* Returns the centroids for each labeled region. (ContainerType_Vector_TcVnPoint2_LREAL; Non-zero interface pointers are reused.) *)
		nLabels	:	REFERENCE TO DINT;	(* Returns the number of labels *)
		eConnectivity	:	ETcVnPixelConnectivity;	(* Selects if 4- or 8-way pixel connectivity should be used *)
		eLabelType	:	ETcVnElementType;	(* Selects the type of ipLabelImage (only UINT or DINT supported) *)
		eAlgorithm	:	ETcVnConnectedComponentsAlgorithm;	(* Selects the applied algorithm *)
		hrPrev	:	HRESULT;	(* HRESULT indicating the result of previous operations (If SUCCEEDED(hrPrev) equals false, no operation is executed.) *)
	END_VAR

END_FUNCTION

// Functions/Image Analysis/F_VN_CountNonZeroPixels

	{attribute 'TcIecLibraryType'}
	{attribute 'external_name' := 'F_VN_CountNonZeroPixels_GUID_E6F098EE_E799_055F_6983_4C863501FB07'}
	(* Counts the non-zero pixels in a single-channel image (e.g. useful to analyze threshold results). *)
	FUNCTION F_VN_CountNonZeroPixels : HRESULT
	VAR_INPUT
		ipSrcImage	:	ITcVnImage;	(* Source image (1 channel) *)
		nNonZero	:	REFERENCE TO ULINT;	(* Returns the number of non-zero pixels in ipSrcImage *)
		hrPrev	:	HRESULT;	(* HRESULT indicating the result of previous operations (If SUCCEEDED(hrPrev) equals false, no operation is executed.) *)
	END_VAR

END_FUNCTION

// Functions/Image Analysis/F_VN_DistanceTransformation

	{attribute 'TcIecLibraryType'}
	{attribute 'external_name' := 'F_VN_DistanceTransformation_GUID_354DDB2A_76EB_04E5_52FC_F5BF84742D9C'}
	(* Calculates the distance transformation, which is the distance to the closest zero pixel in a binary image. *)
	FUNCTION F_VN_DistanceTransformation : HRESULT
	VAR_INPUT
		ipSrcImage	:	ITcVnImage;	(* Source image (USINT, 1 channel) *)
		ipDestImage	:	REFERENCE TO ITcVnImage;	(* Destination image (REAL, 1 channel. An appropriate destination image will be created if required.) *)
		eDistanceType	:	ETcVnDistanceType;	(* Distance computation method (supported: L1, L2, C) *)
		eMaskSize	:	ETcVnDistanceTransformationMask;	(* Size of the distance transformation mask *)
		hrPrev	:	HRESULT;	(* HRESULT indicating the result of previous operations (If SUCCEEDED(hrPrev) equals false, no operation is executed.) *)
	END_VAR

END_FUNCTION

// Functions/Image Analysis/F_VN_DistanceTransformationExp

	{attribute 'TcIecLibraryType'}
	{attribute 'external_name' := 'F_VN_DistanceTransformationExp_GUID_372A7AC7_4A8F_05CA_6371_34441F33EF8E'}
	(* Calculates the distance transformation, which is the distance to the closest zero pixel in a binary image. Additionally, an image with component labels is created (discrete Voronoi diagram). (expert function) *)
	FUNCTION F_VN_DistanceTransformationExp : HRESULT
	VAR_INPUT
		ipSrcImage	:	ITcVnImage;	(* Source image (USINT, 1 channel) *)
		ipDestImage	:	REFERENCE TO ITcVnImage;	(* Destination image (REAL, 1 channel. An appropriate destination image will be created if required.) *)
		eDistanceType	:	ETcVnDistanceType;	(* Distance computation method (supported: L1, L2, C) *)
		eMaskSize	:	ETcVnDistanceTransformationMask;	(* Size of the distance transformation mask (PRECISE not supported for label computation) *)
		ipDestLabels	:	REFERENCE TO ITcVnImage;	(* Returns the component labels (Discrete Voronoi diagram; DINT, 1 channel. An appropriate image will be created if required.) *)
		eLabelType	:	ETcVnDistanceTransformationLabel;	(* Type of the labels *)
		hrPrev	:	HRESULT;	(* HRESULT indicating the result of previous operations (If SUCCEEDED(hrPrev) equals false, no operation is executed.) *)
	END_VAR

END_FUNCTION

// Functions/Image Analysis/F_VN_GetConnectedComponent

	{attribute 'TcIecLibraryType'}
	{attribute 'external_name' := 'F_VN_GetConnectedComponent_GUID_5955EA36_3367_0589_4B62_73755453AA06'}
	(* Get the mask image of a connected component from a label image based on the label ID. *)
	FUNCTION F_VN_GetConnectedComponent : HRESULT
	VAR_INPUT
		ipLabelImage	:	ITcVnImage;	(* Image containing labels for each pixel (1 channel DINT or UINT). *)
		nLabelID	:	DINT;	(* Value of the requested label *)
		ipMaskImage	:	REFERENCE TO ITcVnImage;	(* Returns a mask image marking the pixels that belong to the component (1 channel USINT.) *)
		hrPrev	:	HRESULT;	(* HRESULT indicating the result of previous operations (If SUCCEEDED(hrPrev) equals false, no operation is executed.) *)
	END_VAR

END_FUNCTION

// Functions/Image Analysis/F_VN_GetConnectedComponentExp

	{attribute 'TcIecLibraryType'}
	{attribute 'external_name' := 'F_VN_GetConnectedComponentExp_GUID_E0BCC920_AA55_0809_674F_C38AD515A776'}
	(* Get the mask image (and optionally the outer contour) of a connected component from a label image based on the label ID. (expert function) *)
	FUNCTION F_VN_GetConnectedComponentExp : HRESULT
	VAR_INPUT
		ipLabelImage	:	ITcVnImage;	(* Image containing labels for each pixel (1 channel DINT or UINT). *)
		nLabelID	:	DINT;	(* Value of the requested label *)
		ipMaskImage	:	REFERENCE TO ITcVnImage;	(* Returns a mask image marking the pixels that belong to the component (1 channel USINT. Mask is optional, set to 0 if not required.) *)
		ipContourPoints	:	REFERENCE TO ITcVnContainer;	(* Returns the outer contour of the component(ContainerType_Vector_TcVnPoint2_DINT. Contour is optional, set to 0 if not required.) *)
		hrPrev	:	HRESULT;	(* HRESULT indicating the result of previous operations (If SUCCEEDED(hrPrev) equals false, no operation is executed.) *)
	END_VAR

END_FUNCTION

// Functions/Image Analysis/F_VN_ImageAverage

	{attribute 'TcIecLibraryType'}
	{attribute 'external_name' := 'F_VN_ImageAverage_GUID_7615F4B2_9FA7_0757_52BC_A73407141399'}
	(* Computes the (channel-wise) average pixel value of an image. *)
	FUNCTION F_VN_ImageAverage : HRESULT
	VAR_INPUT
		ipSrcImage	:	ITcVnImage;	(* Source image (1 - 4 channels) *)
		aAverage	:	REFERENCE TO TcVnVector4_LREAL;	(* Returns the (channel-wise) average pixel value of ipSrcImage *)
		hrPrev	:	HRESULT;	(* HRESULT indicating the result of previous operations (If SUCCEEDED(hrPrev) equals false, no operation is executed.) *)
	END_VAR

END_FUNCTION

// Functions/Image Analysis/F_VN_ImageAverageExp

	{attribute 'TcIecLibraryType'}
	{attribute 'external_name' := 'F_VN_ImageAverageExp_GUID_B6431E06_66F0_0FF2_7333_BA8AC1368AE2'}
	(* Computes the (channel-wise) average pixel value of an image. (expert function) *)
	FUNCTION F_VN_ImageAverageExp : HRESULT
	VAR_INPUT
		ipSrcImage	:	ITcVnImage;	(* Source image (1 - 4 channels) *)
		aAverage	:	REFERENCE TO TcVnVector4_LREAL;	(* Returns the (channel-wise) average pixel value of ipSrcImage *)
		ipMask	:	ITcVnImage;	(* Mask of type USINT (1 channel) *)
		hrPrev	:	HRESULT;	(* HRESULT indicating the result of previous operations (If SUCCEEDED(hrPrev) equals false, no operation is executed.) *)
	END_VAR

END_FUNCTION

// Functions/Image Analysis/F_VN_ImageAverageStdDev

	{attribute 'TcIecLibraryType'}
	{attribute 'external_name' := 'F_VN_ImageAverageStdDev_GUID_41D1F46B_D752_01BB_5762_D3B2CA627AAD'}
	(* Computes the (channel-wise) average pixel value and the corresponding standard deviation of an image. *)
	FUNCTION F_VN_ImageAverageStdDev : HRESULT
	VAR_INPUT
		ipSrcImage	:	ITcVnImage;	(* Source image (1 - 4 channels) *)
		aAverage	:	REFERENCE TO TcVnVector4_LREAL;	(* Returns the (channel-wise) average pixel value of ipSrcImage *)
		aStdDev	:	REFERENCE TO TcVnVector4_LREAL;	(* Returns the (channel-wise) pixel value standard deviation of ipSrcImage *)
		hrPrev	:	HRESULT;	(* HRESULT indicating the result of previous operations (If SUCCEEDED(hrPrev) equals false, no operation is executed.) *)
	END_VAR

END_FUNCTION

// Functions/Image Analysis/F_VN_ImageAverageStdDevExp

	{attribute 'TcIecLibraryType'}
	{attribute 'external_name' := 'F_VN_ImageAverageStdDevExp_GUID_0EFC33AA_7F58_012E_7332_63C5E3F3159A'}
	(* Computes the (channel-wise) average pixel value and the corresponding standard deviation of an image. (expert function) *)
	FUNCTION F_VN_ImageAverageStdDevExp : HRESULT
	VAR_INPUT
		ipSrcImage	:	ITcVnImage;	(* Source image (1 - 4 channels) *)
		aAverage	:	REFERENCE TO TcVnVector4_LREAL;	(* Returns the (channel-wise) average pixel value of ipSrcImage *)
		aStdDev	:	REFERENCE TO TcVnVector4_LREAL;	(* Returns the (channel-wise) pixel value standard deviation of ipSrcImage *)
		ipMask	:	ITcVnImage;	(* Mask of type USINT (1 channel) *)
		hrPrev	:	HRESULT;	(* HRESULT indicating the result of previous operations (If SUCCEEDED(hrPrev) equals false, no operation is executed.) *)
	END_VAR

END_FUNCTION

// Functions/Image Analysis/F_VN_ImageCenterOfMass

	{attribute 'TcIecLibraryType'}
	{attribute 'external_name' := 'F_VN_ImageCenterOfMass_GUID_6A0804AA_02B0_0194_6095_324ABB44E3F8'}
	(* Computes the center of mass of an image. *)
	FUNCTION F_VN_ImageCenterOfMass : HRESULT
	VAR_INPUT
		ipSrcImage	:	ITcVnImage;	(* Source image (1 channel) *)
		aCenterOfMass	:	REFERENCE TO TcVnPoint2_LREAL;	(* Returns the center of mass of the image *)
		hrPrev	:	HRESULT;	(* HRESULT indicating the result of previous operations (If SUCCEEDED(hrPrev) equals false, no operation is executed.) *)
	END_VAR

END_FUNCTION

// Functions/Image Analysis/F_VN_ImageCenterOfMassExp

	{attribute 'TcIecLibraryType'}
	{attribute 'external_name' := 'F_VN_ImageCenterOfMassExp_GUID_D189A05F_59EB_01BB_7282_50120F32E617'}
	(* Computes the center of mass of an image. *)
	FUNCTION F_VN_ImageCenterOfMassExp : HRESULT
	VAR_INPUT
		ipSrcImage	:	ITcVnImage;	(* Source image (1 channel) *)
		aCenterOfMass	:	REFERENCE TO TcVnPoint2_LREAL;	(* Returns the center of mass of the image *)
		ipMask	:	ITcVnImage;	(* Optional mask (1 channel of type USINT, same width and height as ipSrcImage) *)
		hrPrev	:	HRESULT;	(* HRESULT indicating the result of previous operations (If SUCCEEDED(hrPrev) equals false, no operation is executed.) *)
	END_VAR

END_FUNCTION

// Functions/Image Analysis/F_VN_ImageMedian

	{attribute 'TcIecLibraryType'}
	{attribute 'external_name' := 'F_VN_ImageMedian_GUID_7C9EF36F_CB9E_0D96_5CB9_E5D78F1A06F9'}
	(* Computes the (approximated, channel-wise) median pixel value of an image. *)
	FUNCTION F_VN_ImageMedian : HRESULT
	VAR_INPUT
		ipSrcImage	:	ITcVnImage;	(* Source image (1 - 4 channels) *)
		aMedian	:	REFERENCE TO TcVnVector4_LREAL;	(* Returns the (approximated, channel-wise) median pixel value of ipSrcImage *)
		hrPrev	:	HRESULT;	(* HRESULT indicating the result of previous operations (If SUCCEEDED(hrPrev) equals false, no operation is executed.) *)
	END_VAR

END_FUNCTION

// Functions/Image Analysis/F_VN_ImageMedianExp

	{attribute 'TcIecLibraryType'}
	{attribute 'external_name' := 'F_VN_ImageMedianExp_GUID_FC58A4FB_0C98_08A6_7545_CC09B54A3632'}
	(* Computes the (approximated, channel-wise) median pixel value of an image. (expert function) *)
	FUNCTION F_VN_ImageMedianExp : HRESULT
	VAR_INPUT
		ipSrcImage	:	ITcVnImage;	(* Source image (1 - 4 channels) *)
		aMedian	:	REFERENCE TO TcVnVector4_LREAL;	(* Returns the (approximated, channel-wise) median pixel value of ipSrcImage *)
		ipMask	:	ITcVnImage;	(* Mask of type USINT (1 channel) *)
		hrPrev	:	HRESULT;	(* HRESULT indicating the result of previous operations (If SUCCEEDED(hrPrev) equals false, no operation is executed.) *)
	END_VAR

END_FUNCTION

// Functions/Image Analysis/F_VN_ImageMoments

	{attribute 'TcIecLibraryType'}
	{attribute 'external_name' := 'F_VN_ImageMoments_GUID_6E8223A9_2B87_04B0_5702_39F5F3BF85AD'}
	(* Computes the spatial moments, the central moments, and the central normalized moments of an image up to the third order. *)
	FUNCTION F_VN_ImageMoments : HRESULT
	VAR_INPUT
		ipImage	:	ITcVnImage;	(* Source image (1 channel, elements of type USINT or REAL) *)
		stMoments	:	REFERENCE TO TcVnMoments;	(* Returns a struct containing the moments *)
		bBinaryImage	:	BOOL;	(* If true, all non-zero pixels are treated as ones *)
		hrPrev	:	HRESULT;	(* HRESULT indicating the result of previous operations (If SUCCEEDED(hrPrev) equals false, no operation is executed.) *)
	END_VAR

END_FUNCTION

// Functions/Image Analysis/F_VN_MaxPixelValue

	{attribute 'TcIecLibraryType'}
	{attribute 'external_name' := 'F_VN_MaxPixelValue_GUID_B9C7D79D_E70F_0530_65BE_F053EFD3111D'}
	(* Finds the maximum pixel value in an image (1 - 4 channels supported). *)
	FUNCTION F_VN_MaxPixelValue : HRESULT
	VAR_INPUT
		ipImage	:	ITcVnImage;	(* Source image *)
		aMaxValue	:	REFERENCE TO TcVnVector4_LREAL;	(* Returns the maximum pixel value *)
		aPosition	:	REFERENCE TO TcVnPoint2_DINT;	(* Returns the first found position of aMaxValue *)
		hrPrev	:	HRESULT;	(* HRESULT indicating the result of previous operations (If SUCCEEDED(hrPrev) equals false, no operation is executed.) *)
	END_VAR

END_FUNCTION

// Functions/Image Analysis/F_VN_MaxPixelValueExp

	{attribute 'TcIecLibraryType'}
	{attribute 'external_name' := 'F_VN_MaxPixelValueExp_GUID_951C3F76_63F2_0CD0_6E7E_F8A0279ECED0'}
	(* Finds the maximum pixel value in an image (1 - 4 channels supported). (expert function) *)
	FUNCTION F_VN_MaxPixelValueExp : HRESULT
	VAR_INPUT
		ipImage	:	ITcVnImage;	(* Source image *)
		aMaxValue	:	REFERENCE TO TcVnVector4_LREAL;	(* Returns the maximum pixel value *)
		aPosition	:	REFERENCE TO TcVnPoint2_DINT;	(* Returns the first found position of aMaxValue (not supported for multi-channel images with ELEMENTWISE) *)
		ipMask	:	ITcVnImage;	(* Optional mask to specify which pixel positions are considered (USINT, set parameter to 0 if not required) *)
		eVectorCompareMethod	:	ETcVnVectorCompareMethod;	(* Select a vector compare method for multi-channel images *)
		hrPrev	:	HRESULT;	(* HRESULT indicating the result of previous operations (If SUCCEEDED(hrPrev) equals false, no operation is executed.) *)
	END_VAR

END_FUNCTION

// Functions/Image Analysis/F_VN_MinPixelValue

	{attribute 'TcIecLibraryType'}
	{attribute 'external_name' := 'F_VN_MinPixelValue_GUID_D42B4D94_34B8_0C1D_424F_EFC472F1C288'}
	(* Finds the minimum pixel value in an image (1 - 4 channels supported). *)
	FUNCTION F_VN_MinPixelValue : HRESULT
	VAR_INPUT
		ipImage	:	ITcVnImage;	(* Source image *)
		aMinValue	:	REFERENCE TO TcVnVector4_LREAL;	(* Returns the minimum pixel value *)
		aPosition	:	REFERENCE TO TcVnPoint2_DINT;	(* Returns the first found position of aMinValue *)
		hrPrev	:	HRESULT;	(* HRESULT indicating the result of previous operations (If SUCCEEDED(hrPrev) equals false, no operation is executed.) *)
	END_VAR

END_FUNCTION

// Functions/Image Analysis/F_VN_MinPixelValueExp

	{attribute 'TcIecLibraryType'}
	{attribute 'external_name' := 'F_VN_MinPixelValueExp_GUID_0C598682_7559_0D0E_76DD_1010EDA6D9AC'}
	(* Finds the minimum pixel value in an image (1 - 4 channels supported). (expert function) *)
	FUNCTION F_VN_MinPixelValueExp : HRESULT
	VAR_INPUT
		ipImage	:	ITcVnImage;	(* Source image *)
		aMinValue	:	REFERENCE TO TcVnVector4_LREAL;	(* Returns the minimum pixel value *)
		aPosition	:	REFERENCE TO TcVnPoint2_DINT;	(* Returns the first found position of aMinValue (not supported for multi-channel images with ELEMENTWISE) *)
		ipMask	:	ITcVnImage;	(* Optional mask to specify which pixel positions are considered (USINT, set parameter to 0 if not required) *)
		eVectorCompareMethod	:	ETcVnVectorCompareMethod;	(* Select a vector compare method for multi-channel images *)
		hrPrev	:	HRESULT;	(* HRESULT indicating the result of previous operations (If SUCCEEDED(hrPrev) equals false, no operation is executed.) *)
	END_VAR

END_FUNCTION

// Functions/Image Analysis/F_VN_RegionOrientation

	{attribute 'TcIecLibraryType'}
	{attribute 'external_name' := 'F_VN_RegionOrientation_GUID_B8526065_FC69_0D8D_4E54_EAF98F2623AD'}
	(* Calculate the orientation of a region based on a binary image that contains a non zero value for every pixel in that region. *)
	FUNCTION F_VN_RegionOrientation : HRESULT
	VAR_INPUT
		ipSrcImage	:	ITcVnImage;	(* Source image (1 channel, binary). *)
		stOrientation	:	REFERENCE TO TcVnRotatedRectangle;	(* Resulting rotated rectangle, containig center of mass, lenghts of axes, and rotation angle of the region in clockwise direction. *)
		hrPrev	:	HRESULT;	(* HRESULT indicating the result of previous operations (If SUCCEEDED(hrPrev) equals false, no operation is executed.) *)
	END_VAR

END_FUNCTION

// Functions/Image Analysis/F_VN_RegionOrientationExp

	{attribute 'TcIecLibraryType'}
	{attribute 'external_name' := 'F_VN_RegionOrientationExp_GUID_A5E7964B_98E9_03C8_5AB5_6B36AB660D83'}
	(* Calculate the orientation of a region based on a binary image that contains a non zero value for every pixel in that region. (expert function) *)
	FUNCTION F_VN_RegionOrientationExp : HRESULT
	VAR_INPUT
		ipSrcImage	:	ITcVnImage;	(* Source image (1 channel, binary) *)
		stOrientation	:	REFERENCE TO TcVnRotatedRectangle;	(* Resulting rotated rectangle, containig center of mass, lenghts of axes, and rotation angle of the region in clockwise direction. *)
		eMethod	:	ETcVnOrientationMethod;	(* Method for calculating the orientation. *)
		hrPrev	:	HRESULT;	(* HRESULT indicating the result of previous operations (If SUCCEEDED(hrPrev) equals false, no operation is executed.) *)
	END_VAR

END_FUNCTION

// Functions/Measurement/F_VN_AdjustSearchWindowOrientationToLinearEdge

	{attribute 'TcIecLibraryType'}
	{attribute 'external_name' := 'F_VN_AdjustSearchWindowOrientationToLinearEdge_GUID_5C77A53D_4CA8_01FC_5A34_A8F8EC7AB5EB'}
	(* Adjust the search window to be orthogonal to a linear edge. Might be helpful before calling edge localization and distance measurement functions that rely on the search window. *)
	FUNCTION F_VN_AdjustSearchWindowOrientationToLinearEdge : HRESULT
	VAR_INPUT
		ipSrcImage	:	ITcVnImage;	(* Source image *)
		aStartPoint	:	REFERENCE TO TcVnPoint2_REAL;	(* Position from which to start the search process (in the direction of aEndPoint), which is not changed *)
		aEndPoint	:	REFERENCE TO TcVnPoint2_REAL;	(* Position where the search process ends, which is adjusted by this function *)
		eEdgeDirection	:	ETcVnEdgeDirection;	(* Specification of the edge direction to search for *)
		fMinStrength	:	REAL;	(* Specification of the minimum strength (intensity difference) of the edge to search for *)
		nMaxThickness	:	UDINT;	(* Specification of the maximum thickness of the edge to search for, which means fMinStrength must be reached within nMaxThickness pixels *)
		nSearchLines	:	UDINT;	(* Width of the search window, i.e. the number of search lines (3, 5, 7, ...), centered around the line specified by aStartPoint and aEndPoint *)
		hrPrev	:	HRESULT;	(* HRESULT indicating the result of previous operations (If SUCCEEDED(hrPrev) equals false, no operation is executed.) *)
	END_VAR

END_FUNCTION

// Functions/Measurement/F_VN_ClosestPointsBF

	{attribute 'TcIecLibraryType'}
	{attribute 'external_name' := 'F_VN_ClosestPointsBF_GUID_EFFBFC09_2B3A_0DEF_6691_F3B4257278E8'}
	(* Find the closest distance between two 2d point sets of the same type, using a brute force approach. *)
	FUNCTION F_VN_ClosestPointsBF : HRESULT
	VAR_INPUT
		ipPointSet1	:	ITcVnContainer;	(* Container with 1st set of 2d points *)
		ipPointSet2	:	ITcVnContainer;	(* Container with 2nd set of 2d points *)
		fMinDist	:	REFERENCE TO LREAL;	(* Returns the minimum distance between 2 points of the different point sets *)
		aPoint1	:	REFERENCE TO TcVnPoint2_LREAL;	(* Returns the point out of ipPointSet1, for which fMinDist is achieved *)
		aPoint2	:	REFERENCE TO TcVnPoint2_LREAL;	(* Returns the point out of ipPointSet2, for which fMinDist is achieved *)
		hrPrev	:	HRESULT;	(* HRESULT indicating the result of previous operations (If SUCCEEDED(hrPrev) equals false, no operation is executed.) *)
	END_VAR

END_FUNCTION

// Functions/Measurement/F_VN_LocateCircularArc

	{attribute 'TcIecLibraryType'}
	{attribute 'external_name' := 'F_VN_LocateCircularArc_GUID_4B160743_5A6A_0C76_574A_D8CADE5C3433'}
	(* Locate a circular arc, using an interpolation method. *)
	FUNCTION F_VN_LocateCircularArc : HRESULT
	VAR_INPUT
		ipSrcImage	:	ITcVnImage;	(* Source image (1 channel) *)
		stCircularArc	:	REFERENCE TO TcVnCircularArc;	(* Returns the circular arc parameters *)
		aCenter	:	REFERENCE TO TcVnPoint2_REAL;	(* Input estimated circle center (only used as a starting point to search for the circle contour, not used for the circle center estimation) *)
		fSearchRadius	:	REAL;	(* Input search radius (starting from aCenter, should be greater than the actual circle radius but aCenter + fSearchRadius should be within the image borders) *)
		fArcDirectionRad	:	LREAL;	(* Input search starting direction in radian. Valid range is [-pi, +pi], where right is 0 rad, top is -pi/2 rad and bottom +pi/2 rad. The circular arc should at least be valid in range fArcDirectionRad +- 0.4 rad. *)
		eEdgeDirection	:	ETcVnEdgeDirection;	(* Specification of the edge direction to search for *)
		fMinStrength	:	REAL;	(* Specification of the minimum strength (intensity difference) of the edge to search for *)
		hrPrev	:	HRESULT;	(* HRESULT indicating the result of previous operations (If SUCCEEDED(hrPrev) equals false, no operation is executed.) *)
	END_VAR

END_FUNCTION

// Functions/Measurement/F_VN_LocateCircularArcExp

	{attribute 'TcIecLibraryType'}
	{attribute 'external_name' := 'F_VN_LocateCircularArcExp_GUID_C5189D0A_16D2_0006_627A_84F75A1C244A'}
	(* Locate a circular arc. (expert function) *)
	FUNCTION F_VN_LocateCircularArcExp : HRESULT
	VAR_INPUT
		ipSrcImage	:	ITcVnImage;	(* Source image (1 channel) *)
		stCircularArc	:	REFERENCE TO TcVnCircularArc;	(* Returns the circular arc parameters *)
		aCenter	:	REFERENCE TO TcVnPoint2_REAL;	(* Input estimated circle center (only used as a starting point to search for the circle contour, not used for the circle center estimation) *)
		fSearchRadius	:	REAL;	(* Input search radius (starting from aCenter, should be greater than the actual circle radius but aCenter + fSearchRadius should be within the image borders) *)
		fArcDirectionRad	:	LREAL;	(* Input search starting direction in radian. Valid range is [-pi, +pi], where right is 0 rad, top is -pi/2 rad and bottom +pi/2 rad. The circular arc should at least be valid in range fArcDirectionRad +- 4 * fAngleStepRad) *)
		eEdgeDirection	:	ETcVnEdgeDirection;	(* Specification of the edge direction to search for *)
		fMinStrength	:	REAL;	(* Specification of the minimum strength (intensity difference) of the edge to search for *)
		fAngleStepRad	:	LREAL;	(* Search step in rad (should be chosen so that about 20 - 60 steps are available for the whole arc. In most cases 0.1 rad (5.7 deg) is a good value) *)
		nMaxThickness	:	UDINT;	(* Specification of the maximum thickness of the edge to search for, which means fMinStrength must be reached within nMaxThickness pixels *)
		bInvertSearchDirection	:	BOOL;	(* If true, the search starts from outside the circular arc in direction of the center *)
		nSubpixelsIterations	:	UDINT;	(* Specifies the number of subpixels (for INTERPOLATION, 10 - 20 usually is sufficient) or maximum number of iterations for optimizing the parameters (for APPROX_ERF and APPROX_GAUSSIAN, 50 - 100 usually is sufficient) *)
		fApproxPrecision	:	REAL;	(* Specifies the approximation precision for APPROX_ERF and APPROX_GAUSSIAN (0.001 usually is sufficient, unused for INTERPOLATION) *)
		eAlgorithm	:	ETcVnEdgeDetectionAlgorithm;	(* Selection of the edge detection algorithm *)
		ipContourPoints	:	REFERENCE TO ITcVnContainer;	(* Returns the subpixel accurate contour (optional, set to 0 if not required; ContainerType_Vector_TcVnPoint2_REAL; Non-zero interface pointers are reused.) *)
		hrPrev	:	HRESULT;	(* HRESULT indicating the result of previous operations (If SUCCEEDED(hrPrev) equals false, no operation is executed.) *)
	END_VAR

END_FUNCTION

// Functions/Measurement/F_VN_LocateEdge

	{attribute 'TcIecLibraryType'}
	{attribute 'external_name' := 'F_VN_LocateEdge_GUID_7AEA2696_415F_03B8_78F1_362B79AF09CF'}
	(* Locate the points of the first occuring edge inside a specified search window, using an interpolation method. *)
	FUNCTION F_VN_LocateEdge : HRESULT
	VAR_INPUT
		ipSrcImage	:	ITcVnImage;	(* Source image (1 channel) *)
		ipEdgePoints	:	REFERENCE TO ITcVnContainer;	(* Returns the detected edge points (ContainerType_Vector_TcVnPoint2_REAL) *)
		aStartPoint	:	REFERENCE TO TcVnPoint2_REAL;	(* Position from which to start the search process (in the direction of aEndPoint) *)
		aEndPoint	:	REFERENCE TO TcVnPoint2_REAL;	(* Position where the search process ends *)
		eEdgeDirection	:	ETcVnEdgeDirection;	(* Specification of the edge direction to search for *)
		fMinStrength	:	REAL;	(* Specification of the minimum strength (intensity difference) of the edge to search for *)
		nSearchLines	:	UDINT;	(* Width of the search window, i.e. the number of search lines (1, 3, 5, 7, ...), centered around the line specified by aStartPoint and aEndPoint *)
		hrPrev	:	HRESULT;	(* HRESULT indicating the result of previous operations (If SUCCEEDED(hrPrev) equals false, no operation is executed.) *)
	END_VAR
	VAR_OUTPUT
		fAvgStrength	:	REAL;	(* Returns the average strength of the detected edge *)
	END_VAR

END_FUNCTION

// Functions/Measurement/F_VN_LocateEdgeExp

	{attribute 'TcIecLibraryType'}
	{attribute 'external_name' := 'F_VN_LocateEdgeExp_GUID_6609D35D_3450_034C_4CE8_6E885402E8CA'}
	(* Locate the points of the first occuring edge inside a specified search window with subpixel accuracy. (expert function) *)
	FUNCTION F_VN_LocateEdgeExp : HRESULT
	VAR_INPUT
		ipSrcImage	:	ITcVnImage;	(* Source image (1 channel) *)
		ipEdgePoints	:	REFERENCE TO ITcVnContainer;	(* Returns the detected edge points (ContainerType_Vector_TcVnPoint2_REAL) *)
		aStartPoint	:	REFERENCE TO TcVnPoint2_REAL;	(* Position from which to start the search process (in the direction of aEndPoint) *)
		aEndPoint	:	REFERENCE TO TcVnPoint2_REAL;	(* Position where the search process ends *)
		eEdgeDirection	:	ETcVnEdgeDirection;	(* Specification of the edge direction to search for *)
		fMinStrength	:	REAL;	(* Specification of the minimum strength (intensity difference) of the edge to search for *)
		nSearchLines	:	UDINT;	(* Width of the search window, i.e. the number of search lines (1, 3, 5, 7, ...), centered around the line specified by aStartPoint and aEndPoint *)
		fSearchLineDist	:	REAL;	(* Distance between the search lines in pixels (> 0) *)
		nMaxThickness	:	UDINT;	(* Specification of the maximum thickness of the edge to search for, which means fMinStrength must be reached within nMaxThickness pixels *)
		nSubpixelsIterations	:	UDINT;	(* Specifies the number of subpixels (for INTERPOLATION, 10 - 20 usually is sufficient) or maximum number of iterations for optimizing the parameters (for APPROX_ERF and APPROX_GAUSSIAN, 50 - 100 usually is sufficient) *)
		fApproxPrecision	:	REAL;	(* Specifies the approximation precision for APPROX_ERF and APPROX_GAUSSIAN (0.001 usually is sufficient, unused for INTERPOLATION) *)
		eAlgorithm	:	ETcVnEdgeDetectionAlgorithm;	(* Selection of the edge detection algorithm *)
		hrPrev	:	HRESULT;	(* HRESULT indicating the result of previous operations (If SUCCEEDED(hrPrev) equals false, no operation is executed.) *)
	END_VAR
	VAR_OUTPUT
		fAvgStrength	:	REAL;	(* Returns the average strength of the detected edge *)
	END_VAR

END_FUNCTION

// Functions/Measurement/F_VN_LocateEdges

	{attribute 'TcIecLibraryType'}
	{attribute 'external_name' := 'F_VN_LocateEdges_GUID_0142F338_2E21_044D_72FD_D35AD0F5F3A7'}
	(* Locate the points of multiple occuring edges inside a specified search window, using an interpolation method. *)
	FUNCTION F_VN_LocateEdges : HRESULT
	VAR_INPUT
		ipSrcImage	:	ITcVnImage;	(* Source image (1 channel) *)
		ipEdgePoints	:	REFERENCE TO ITcVnContainer;	(* Returns the detected edge points (ContainerType_Vector_Vector_TcVnPoint2_REAL) *)
		aStartPoint	:	REFERENCE TO TcVnPoint2_REAL;	(* Position from which to start the search process (in the direction of aEndPoint) *)
		aEndPoint	:	REFERENCE TO TcVnPoint2_REAL;	(* Position where the search process ends *)
		nNumEdges	:	UDINT;	(* The (maximum) number of edges to search for *)
		eEdgeDirection	:	ETcVnEdgeDirection;	(* Specification of the edge direction to search for *)
		bAlternateDirection	:	BOOL;	(* If true, eEdgeDirection is alternated after each detected edge. Else, only edges with eEdgeDirection are searched for. *)
		fMinStrength	:	REAL;	(* Specification of the minimum strength (intensity difference) of the edge to search for *)
		nSearchLines	:	UDINT;	(* Width of the search window, i.e. the number of search lines (1, 3, 5, 7, ...), centered around the line specified by aStartPoint and aEndPoint *)
		hrPrev	:	HRESULT;	(* HRESULT indicating the result of previous operations (If SUCCEEDED(hrPrev) equals false, no operation is executed.) *)
	END_VAR
	VAR_OUTPUT
		fAvgStrength	:	REAL;	(* Returns the average strength of the detected edges *)
	END_VAR

END_FUNCTION

// Functions/Measurement/F_VN_LocateEdgesExp

	{attribute 'TcIecLibraryType'}
	{attribute 'external_name' := 'F_VN_LocateEdgesExp_GUID_3324BCF4_945E_0380_480B_051B8267924A'}
	(* Locate the points of multiple occuring edges inside a specified search window with subpixel accuracy. (expert function) *)
	FUNCTION F_VN_LocateEdgesExp : HRESULT
	VAR_INPUT
		ipSrcImage	:	ITcVnImage;	(* Source image (1 channel) *)
		ipEdgePoints	:	REFERENCE TO ITcVnContainer;	(* Returns the detected edge points (ContainerType_Vector_Vector_TcVnPoint2_REAL) *)
		aStartPoint	:	REFERENCE TO TcVnPoint2_REAL;	(* Position from which to start the search process (in the direction of aEndPoint) *)
		aEndPoint	:	REFERENCE TO TcVnPoint2_REAL;	(* Position where the search process ends *)
		nNumEdges	:	UDINT;	(* The (maximum) number of edges to search for *)
		eEdgeDirection	:	ETcVnEdgeDirection;	(* Specification of the edge direction to search for *)
		bAlternateDirection	:	BOOL;	(* If true, eEdgeDirection is alternated after each detected edge. Else, only edges with eEdgeDirection are searched for. *)
		fMinStrength	:	REAL;	(* Specification of the minimum strength (intensity difference) of the edge to search for *)
		nSearchLines	:	UDINT;	(* Width of the search window, i.e. the number of search lines (1, 3, 5, 7, ...), centered around the line specified by aStartPoint and aEndPoint *)
		fSearchLineDist	:	REAL;	(* Distance between the search lines in pixels (> 0) *)
		nMaxThickness	:	UDINT;	(* Specification of the maximum thickness of the edge to search for, which means fMinStrength must be reached within nMaxThickness pixels *)
		nSubpixelsIterations	:	UDINT;	(* Specifies the number of subpixels (for INTERPOLATION, 10 - 20 usually is sufficient) or maximum number of iterations for optimizing the parameters (for APPROX_ERF and APPROX_GAUSSIAN, 50 - 100 usually is sufficient) *)
		fApproxPrecision	:	REAL;	(* Specifies the approximation precision for APPROX_ERF and APPROX_GAUSSIAN (0.001 usually is sufficient, unused for INTERPOLATION) *)
		eAlgorithm	:	ETcVnEdgeDetectionAlgorithm;	(* Selection of the edge detection algorithm *)
		hrPrev	:	HRESULT;	(* HRESULT indicating the result of previous operations (If SUCCEEDED(hrPrev) equals false, no operation is executed.) *)
	END_VAR
	VAR_OUTPUT
		fAvgStrength	:	REAL;	(* Returns the average strength of the detected edges *)
	END_VAR

END_FUNCTION

// Functions/Measurement/F_VN_LocateEllipse

	{attribute 'TcIecLibraryType'}
	{attribute 'external_name' := 'F_VN_LocateEllipse_GUID_6ADC5225_14AE_0582_41D5_0CCF85C7FAE8'}
	(* Locate an ellipse, using an interpolation method for locating the edges. *)
	FUNCTION F_VN_LocateEllipse : HRESULT
	VAR_INPUT
		ipSrcImage	:	ITcVnImage;	(* Source image (1 channel) *)
		stEllipse	:	REFERENCE TO TcVnRotatedRectangle;	(* Returns the detected ellipse *)
		aCenter	:	REFERENCE TO TcVnPoint2_REAL;	(* The expected ellipse center *)
		fSearchRadius	:	REAL;	(* Radius around aCenter to search for edges (aCenter + fSearchRadius in all directions must be inside image borders!) *)
		eEdgeDirection	:	ETcVnEdgeDirection;	(* Specification of the edge direction to search for (from center to outside ellipse) *)
		fMinStrength	:	REAL;	(* Specification of the minimum strength (intensity difference) of the edge to search for *)
		hrPrev	:	HRESULT;	(* HRESULT indicating the result of previous operations (If SUCCEEDED(hrPrev) equals false, no operation is executed.) *)
	END_VAR

END_FUNCTION

// Functions/Measurement/F_VN_LocateEllipseExp

	{attribute 'TcIecLibraryType'}
	{attribute 'external_name' := 'F_VN_LocateEllipseExp_GUID_1DEF14A7_68AF_0AE9_5C75_A1AB2A6416BB'}
	(* Locate an ellipse. (expert function) *)
	FUNCTION F_VN_LocateEllipseExp : HRESULT
	VAR_INPUT
		ipSrcImage	:	ITcVnImage;	(* Source image (1 channel) *)
		stEllipse	:	REFERENCE TO TcVnRotatedRectangle;	(* Returns the detected ellipse *)
		aCenter	:	REFERENCE TO TcVnPoint2_REAL;	(* The expected ellipse center *)
		fSearchRadius	:	REAL;	(* Radius around aCenter to search for edges *)
		eEdgeDirection	:	ETcVnEdgeDirection;	(* Specification of the edge direction to search for (from center to outside ellipse or other way round, if bInvertSearchDirection is true) *)
		fMinStrength	:	REAL;	(* Specification of the minimum strength (intensity difference) of the edge to search for *)
		nMaxThickness	:	UDINT;	(* Specification of the maximum thickness of the edge to search for, which means fMinStrength must be reached within nMaxThickness pixels *)
		bInvertSearchDirection	:	BOOL;	(* If true, the search starts from outside the ellipse in direction of the center *)
		fMinSearchRadius	:	REAL;	(* Radius around aCenter to skip before starting to search for edges (e.g. to save time or if the center contains edges that should be ignored) *)
		nSubpixelsIterations	:	UDINT;	(* Specifies the number of subpixels (for INTERPOLATION, 10 - 20 usually is sufficient) or maximum number of iterations for optimizing the parameters (for APPROX_ERF and APPROX_GAUSSIAN, 50 - 100 usually is sufficient) *)
		nSearchLines	:	UDINT;	(* Specifies the amount of search lines, which are equally distributed in all directions (must be >= 8 and a multiple of 4) *)
		fApproxPrecision	:	REAL;	(* Specifies the approximation precision for APPROX_ERF and APPROX_GAUSSIAN (0.001 usually is sufficient, unused for INTERPOLATION) *)
		eAlgorithm	:	ETcVnEdgeDetectionAlgorithm;	(* Selection of the edge detection algorithm *)
		ipContourPoints	:	REFERENCE TO ITcVnContainer;	(* Returns the subpixel accurate ellipse contour (optional, set to 0 if not required; ContainerType_Vector_TcVnPoint2_REAL; Non-zero interface pointers are reused.) *)
		hrPrev	:	HRESULT;	(* HRESULT indicating the result of previous operations (If SUCCEEDED(hrPrev) equals false, no operation is executed.) *)
	END_VAR

END_FUNCTION

// Functions/Measurement/F_VN_MeasureAngleBetweenEdges

	{attribute 'TcIecLibraryType'}
	{attribute 'external_name' := 'F_VN_MeasureAngleBetweenEdges_GUID_C7CA01DE_E2C7_0950_5155_7639E3398FC3'}
	(* Measure the angle between 2 edges, using an interpolation method. *)
	FUNCTION F_VN_MeasureAngleBetweenEdges : HRESULT
	VAR_INPUT
		ipSrcImage	:	ITcVnImage;	(* Source image (1 channel) *)
		fAngle	:	REFERENCE TO REAL;	(* Returns the angle between the detected edges (radians) *)
		aInnerPoint	:	REFERENCE TO TcVnPoint2_REAL;	(* Position inside the angle to measure, from which to start the edge search process (in the direction of aOuterPoint1 and aOuterPoint2) *)
		aOuterPoint1	:	REFERENCE TO TcVnPoint2_REAL;	(* Position where the search process for edge 1 ends *)
		aOuterPoint2	:	REFERENCE TO TcVnPoint2_REAL;	(* Position where the search process for edge 2 ends *)
		eEdgeDirection	:	ETcVnEdgeDirection;	(* Specification of the edge direction from aInnerPoint to aOuterPoint1 and aOuterPoint2 to search for *)
		fMinStrength	:	REAL;	(* Specification of the minimum strength (intensity difference) of the edge to search for *)
		nSearchLines	:	UDINT;	(* Width of the search windows, i.e. the number of search lines (3, 5, 7, ...), centered around the lines specified by aInnerPoint and aOuterPoint1, aOuterPoint2 *)
		hrPrev	:	HRESULT;	(* HRESULT indicating the result of previous operations (If SUCCEEDED(hrPrev) equals false, no operation is executed.) *)
	END_VAR

END_FUNCTION

// Functions/Measurement/F_VN_MeasureAngleBetweenEdgesExp

